METHOD PUBLIC ClearReference
VAR_INPUT
END_VAR
activeData REF= localData;
SetMemberReference();
END_METHOD

PROPERTY PUBLIC Size : UDINT
GET
Size := SIZEOF(activeData);
END_GET
END_PROPERTY

METHOD FB_init : BOOL
VAR_INPUT
	bInitRetains : BOOL; // if TRUE, the retain variables are initialized (warm start / cold start)
	bInCopyCode : BOOL;  // if TRUE, the instance afterwards gets moved into the copy code (online change)
END_VAR
SetMemberReference();
AddMember('bFilterByArea', _bFilterByArea);
AddMember('bFilterByCircularity', _bFilterByCircularity);
AddMember('bFilterByColor', _bFilterByColor);
AddMember('bFilterByConvexity', _bFilterByConvexity);
AddMember('bFilterByInertia', _bFilterByInertia);
AddMember('fMinArea', _fMinArea);
AddMember('fMaxArea', _fMaxArea);
AddMember('fMinCircularity', _fMinCircularity);
AddMember('fMaxCircularity', _fMaxCircularity);
AddMember('nBlobColor', _nBlobColor);
AddMember('fMinConvexity', _fMinConvexity);
AddMember('fMaxConvexity', _fMaxConvexity);
AddMember('fMinInertiaRatio', _fMinInertiaRatio);
AddMember('fMaxInertiaRatio', _fMaxInertiaRatio);
AddMember('fMinBlobDist', _fMinBlobDist);
AddMember('nMinRepeatability', _nMinRepeatability);
AddMember('fMinThreshold', _fMinThreshold);
AddMember('fMaxThreshold', _fMaxThreshold);
AddMember('fThresholdStep',  _fThresholdStep);
END_METHOD

METHOD PROTECTED SetMemberReference
VAR_INPUT
END_VAR
_bFilterByArea.MakeReferenceTo(activeData.bFilterByArea);
_bFilterByCircularity.MakeReferenceTo(activeData.bFilterByCircularity);
_bFilterByColor.MakeReferenceTo(activeData.bFilterByColor);
_bFilterByConvexity.MakeReferenceTo(activeData.bFilterByConvexity);
_bFilterByInertia.MakeReferenceTo(activeData.bFilterByInertia);
_fMinArea.MakeReferenceTo(activeData.fMinArea);
_fMaxArea.MakeReferenceTo(activeData.fMaxArea);
_fMinCircularity.MakeReferenceTo(activeData.fMinCircularity);
_fMaxCircularity.MakeReferenceTo(activeData.fMaxCircularity);
_nBlobColor.MakeReferenceTo(activeData.nBlobColor);
_fMinConvexity.MakeReferenceTo(activeData.fMinConvexity);
_fMaxConvexity.MakeReferenceTo(activeData.fMaxConvexity);
_fMinInertiaRatio.MakeReferenceTo(activeData.fMinInertiaRatio);
_fMaxInertiaRatio.MakeReferenceTo(activeData.fMaxInertiaRatio);
_fMinBlobDist.MakeReferenceTo(activeData.fMinBlobDist);
_nMinRepeatability.MakeReferenceTo(activeData.nMinRepeatability);
_fMinThreshold.MakeReferenceTo(activeData.fMinThreshold);
_fMaxThreshold.MakeReferenceTo(activeData.fMaxThreshold);
_fThresholdStep.MakeReferenceTo(activeData.fThresholdStep);
END_METHOD

METHOD PUBLIC Clone : I_Datatype
VAR
    pClone : POINTER TO _TcVnParamsSB;
END_VAR
pClone := __NEW(_TcVnParamsSB());
pClone^.Value := Value;
Clone := pClone^;
END_METHOD

PROPERTY PUBLIC Identifier : T_MAXSTRING
GET
Identifier := 'TcVnParamsSB';
END_GET
END_PROPERTY

METHOD PUBLIC MakeReferenceTo
VAR_INPUT
	ReferenceTarget : REFERENCE TO TcVnParamsSB;
END_VAR
activeData REF= ReferenceTarget;
SetMemberReference();
END_METHOD

METHOD TryMakeReferenceTo : BOOL
VAR_INPUT
	Target : I_Datatype;
END_VAR
VAR
	pTargetData : POINTER TO TcVnParamsSB;
END_VAR
IF NOT IsEquivalentTo(Target) THEN
	RETURN;
END_IF

pTargetData := Target.Address;
activeData REF= pTargetData^;
SetMemberReference();
TryMakeReferenceTo := TRUE;
END_METHOD

PROPERTY PUBLIC Value : REFERENCE TO TcVnParamsSB
GET
Value REF= activeData;
END_GET
END_PROPERTY

PROPERTY PUBLIC bFilterByArea : REFERENCE TO _BOOL
GET
bFilterByArea REF= _bFilterByArea;
END_GET
END_PROPERTY

PROPERTY PUBLIC bFilterByCircularity : REFERENCE TO _BOOL
GET
bFilterByCircularity REF= _bFilterByCircularity;
END_GET
END_PROPERTY

PROPERTY PUBLIC bFilterByColor : REFERENCE TO _BOOL
GET
bFilterByColor REF= _bFilterByColor;
END_GET
END_PROPERTY

PROPERTY PUBLIC bFilterByConvexity : REFERENCE TO _BOOL
GET
bFilterByConvexity REF= _bFilterByConvexity;
END_GET
END_PROPERTY

PROPERTY PUBLIC bFilterByInertia : REFERENCE TO _BOOL
GET
bFilterByInertia REF= _bFilterByInertia;
END_GET
END_PROPERTY

PROPERTY PUBLIC fMaxArea : REFERENCE TO _REAL
GET
fMaxArea REF= _fMaxArea;
END_GET
END_PROPERTY

PROPERTY PUBLIC fMaxCircularity : REFERENCE TO _REAL
GET
fMaxCircularity REF= _fMaxCircularity;
END_GET
END_PROPERTY

PROPERTY PUBLIC fMaxConvexity : REFERENCE TO _REAL
GET
fMaxConvexity REF= _fMaxConvexity;
END_GET
END_PROPERTY

PROPERTY PUBLIC fMaxInertiaRatio : REFERENCE TO _REAL
GET
fMaxInertiaRatio REF= _fMaxInertiaRatio;
END_GET
END_PROPERTY

PROPERTY PUBLIC fMaxThreshold : REFERENCE TO _REAL
GET
fMaxThreshold REF= _fMaxThreshold;
END_GET
END_PROPERTY

PROPERTY PUBLIC fMinArea : REFERENCE TO _REAL
GET
fMinArea REF= _fMinArea;
END_GET
END_PROPERTY

PROPERTY PUBLIC fMinBlobDist : REFERENCE TO _REAL
GET
fMinBlobDist REF= _fMinBlobDist;
END_GET
END_PROPERTY

PROPERTY PUBLIC fMinCircularity : REFERENCE TO _REAL
GET
fMinCircularity REF= _fMinCircularity;
END_GET
END_PROPERTY

PROPERTY PUBLIC fMinConvexity : REFERENCE TO _REAL
GET
fMinConvexity REF= _fMinConvexity;
END_GET
END_PROPERTY

PROPERTY PUBLIC fMinInertiaRatio : REFERENCE TO _REAL
GET
fMinInertiaRatio REF= _fMinInertiaRatio;
END_GET
END_PROPERTY

PROPERTY PUBLIC fMinThreshold : REFERENCE TO _REAL
GET
fMinThreshold REF= _fMinThreshold;
END_GET
END_PROPERTY

PROPERTY PUBLIC fThresholdStep : REFERENCE TO _REAL
GET
fThresholdStep REF= _fThresholdStep;
END_GET
END_PROPERTY

PROPERTY PUBLIC nBlobColor : REFERENCE TO _USINT
GET
nBlobColor REF= _nBlobColor;
END_GET
END_PROPERTY

PROPERTY PUBLIC nMinRepeatability : REFERENCE TO _UDINT
GET
nMinRepeatability REF= _nMinRepeatability;
END_GET
END_PROPERTY

END_FUNCTION_BLOCK

// Datatypes/Structs/_TcVnParamsWalshBarcodeDetection
{attribute 'linkalways'}
{attribute 'no_explicit_call' := 'This FB is a CLASS and must be accessed using methods or properties'}
{attribute 'enable_dynamic_creation'}
FUNCTION_BLOCK _TcVnParamsWalshBarcodeDetection EXTENDS StructuredDatatypeBase
VAR
    localData : TcVnParamsWalshBarcodeDetection := (nMaxBarDistance := 8, fMinAspectRatio := 1.0, fMaxAspectRatio := 5.0, nIntensityDifference := 100, nMinArea := -1, nChannelIndex := -1, nWalshFilterNum := 5, fOutlierReductionFactor := 1.0, fBarConnectionFactor := 1.0, fRegionFilterFactor := 1.0, fPostProcessingResizeFactor := 0.5, eInterpolationType := TCVN_IT_BILINEAR);
    activeData : REFERENCE TO TcVnParamsWalshBarcodeDetection REF= localData;
    _nMaxBarDistance : _UDINT(localData.nMaxBarDistance);
    _fMinAspectRatio : _REAL(localData.fMinAspectRatio);
    _fMaxAspectRatio : _REAL(localData.fMaxAspectRatio);
    _nIntensityDifference : _UDINT(localData.nIntensityDifference);
    _nMinArea : _DINT(localData.nMinArea);
    _nChannelIndex : _DINT(localData.nChannelIndex);
    _nWalshFilterNum : _UDINT(localData.nWalshFilterNum);
    _fOutlierReductionFactor : _REAL(localData.fOutlierReductionFactor);
    _fBarConnectionFactor : _REAL(localData.fBarConnectionFactor);
    _fRegionFilterFactor : _REAL(localData.fRegionFilterFactor);
    _fPostProcessingResizeFactor : _REAL(localData.fPostProcessingResizeFactor);
    _eInterpolationType : _ETcVnInterpolationType(localData.eInterpolationType);
END_VAR

PROPERTY PUBLIC Address : PVOID
GET
Address := ADR(activeData);
END_GET
END_PROPERTY

METHOD PUBLIC ClearReference
VAR_INPUT
END_VAR
activeData REF= localData;
SetMemberReference();
END_METHOD

PROPERTY PUBLIC Size : UDINT
GET
Size := SIZEOF(activeData);
END_GET
END_PROPERTY

METHOD FB_init : BOOL
VAR_INPUT
	bInitRetains : BOOL; // if TRUE, the retain variables are initialized (warm start / cold start)
	bInCopyCode : BOOL;  // if TRUE, the instance afterwards gets moved into the copy code (online change)
END_VAR
SetMemberReference();
AddMember('nMaxBarDistance', _nMaxBarDistance);
AddMember('fMinAspectRatio', _fMinAspectRatio);
AddMember('fMaxAspectRatio', _fMaxAspectRatio);
AddMember('nIntensityDifference', _nIntensityDifference);
AddMember('nMinArea', _nMinArea);
AddMember('nChannelIndex', _nChannelIndex);
AddMember('nWalshFilterNum', _nWalshFilterNum);
AddMember('fOutlierReductionFactor', _fOutlierReductionFactor);
AddMember('fBarConnectionFactor', _fBarConnectionFactor);
AddMember('fRegionFilterFactor', _fRegionFilterFactor);
AddMember('fPostProcessingResizeFactor', _fPostProcessingResizeFactor);
AddMember('eInterpolationType', _eInterpolationType);
END_METHOD

METHOD PROTECTED SetMemberReference
VAR_INPUT
END_VAR
_nMaxBarDistance.MakeReferenceTo(activeData.nMaxBarDistance);
_fMinAspectRatio.MakeReferenceTo(activeData.fMinAspectRatio);
_fMaxAspectRatio.MakeReferenceTo(activeData.fMaxAspectRatio);
_nIntensityDifference.MakeReferenceTo(activeData.nIntensityDifference);
_nMinArea.MakeReferenceTo(activeData.nMinArea);
_nChannelIndex.MakeReferenceTo(activeData.nChannelIndex);
_nWalshFilterNum.MakeReferenceTo(activeData.nWalshFilterNum);
_fOutlierReductionFactor.MakeReferenceTo(activeData.fOutlierReductionFactor);
_fBarConnectionFactor.MakeReferenceTo(activeData.fBarConnectionFactor);
_fRegionFilterFactor.MakeReferenceTo(activeData.fRegionFilterFactor);
_fPostProcessingResizeFactor.MakeReferenceTo(activeData.fPostProcessingResizeFactor);
_eInterpolationType.MakeReferenceTo(activeData.eInterpolationType);
END_METHOD

METHOD PUBLIC Clone : I_Datatype
VAR
    pClone : POINTER TO _TcVnParamsWalshBarcodeDetection;
END_VAR
pClone := __NEW(_TcVnParamsWalshBarcodeDetection);
IF pClone = 0 THEN
    RETURN;
END_IF
pClone^.TryCopyFrom(THIS^);
Clone := pClone^;
END_METHOD

PROPERTY PUBLIC Identifier : T_MAXSTRING
GET
Identifier := 'TcVnParamsWalshBarcodeDetection';
END_GET
END_PROPERTY

METHOD PUBLIC MakeReferenceTo
VAR_INPUT
	ReferenceTarget : REFERENCE TO TcVnParamsWalshBarcodeDetection;
END_VAR
activeData REF= ReferenceTarget;
SetMemberReference();
END_METHOD

METHOD TryMakeReferenceTo : BOOL
VAR_INPUT
	Target : I_Datatype;
END_VAR
VAR
	pTargetData : POINTER TO TcVnParamsWalshBarcodeDetection;
END_VAR
IF NOT IsEquivalentTo(Target) THEN
	RETURN;
END_IF

pTargetData := Target.Address;
activeData REF= pTargetData^;
SetMemberReference();
TryMakeReferenceTo := TRUE;
END_METHOD

PROPERTY PUBLIC Value : REFERENCE TO TcVnParamsWalshBarcodeDetection
GET
Value REF= activeData;
END_GET
END_PROPERTY

PROPERTY PUBLIC eInterpolationType : REFERENCE TO _ETcVnInterpolationType
GET
eInterpolationType REF= _eInterpolationType;
END_GET
END_PROPERTY

PROPERTY PUBLIC fBarConnectionFactor : REFERENCE TO _REAL
GET
fBarConnectionFactor REF= _fBarConnectionFactor;
END_GET
END_PROPERTY

PROPERTY PUBLIC fMaxAspectRatio : REFERENCE TO _REAL
GET
fMaxAspectRatio REF= _fMaxAspectRatio;
END_GET
END_PROPERTY

PROPERTY PUBLIC fMinAspectRatio : REFERENCE TO _REAL
GET
fMinAspectRatio REF= _fMinAspectRatio;
END_GET
END_PROPERTY

PROPERTY PUBLIC fOutlierReductionFactor : REFERENCE TO _REAL
GET
fOutlierReductionFactor REF= _fOutlierReductionFactor;
END_GET
END_PROPERTY

PROPERTY PUBLIC fPostProcessingResizeFactor : REFERENCE TO _REAL
GET
fPostProcessingResizeFactor REF= _fPostProcessingResizeFactor;
END_GET
END_PROPERTY

PROPERTY PUBLIC fRegionFilterFactor : REFERENCE TO _REAL
GET
fRegionFilterFactor REF= _fRegionFilterFactor;
END_GET
END_PROPERTY

PROPERTY PUBLIC nChannelIndex : REFERENCE TO _DINT
GET
nChannelIndex REF= _nChannelIndex;
END_GET
END_PROPERTY

PROPERTY PUBLIC nIntensityDifference : REFERENCE TO _UDINT
GET
nIntensityDifference REF= _nIntensityDifference;
END_GET
END_PROPERTY

PROPERTY PUBLIC nMaxBarDistance : REFERENCE TO _UDINT
GET
nMaxBarDistance REF= _nMaxBarDistance;
END_GET
END_PROPERTY

PROPERTY PUBLIC nMinArea : REFERENCE TO _DINT
GET
nMinArea REF= _nMinArea;
END_GET
END_PROPERTY

PROPERTY PUBLIC nWalshFilterNum : REFERENCE TO _UDINT
GET
nWalshFilterNum REF= _nWalshFilterNum;
END_GET
END_PROPERTY

END_FUNCTION_BLOCK

// Datatypes/Structs/_TcVnRectangle_UDINT
{attribute 'linkalways'} 
{attribute 'no_explicit_call' := 'This FB is a CLASS and must be accessed using methods or properties'}
{attribute 'enable_dynamic_creation'}
FUNCTION_BLOCK _TcVnRectangle_UDINT EXTENDS StructuredDatatypeBase
VAR
	localData : TcVnRectangle_UDINT;
	activeData : REFERENCE TO TcVnRectangle_UDINT REF= localData;
	_nX : _UDINT(localData.nX);
	_nY : _UDINT(localData.nY);
    _nWidth : _UDINT(localData.nWidth);
	_nHeight : _UDINT(localData.nHeight);
END_VAR

PROPERTY PUBLIC Address : PVOID
GET
Address := ADR(activeData);
END_GET
END_PROPERTY

METHOD PUBLIC ClearReference
VAR_INPUT
END_VAR
activeData REF= localData;
SetMemberReference();
END_METHOD

PROPERTY PUBLIC Size : UDINT
GET
Size := SIZEOF(activeData);
END_GET
END_PROPERTY

METHOD FB_init : BOOL
VAR_INPUT
	bInitRetains : BOOL; // if TRUE, the retain variables are initialized (warm start / cold start)
	bInCopyCode : BOOL;  // if TRUE, the instance afterwards gets moved into the copy code (online change)
END_VAR
SetMemberReference();
AddMember('nX',_nX);
AddMember('nY',_nY);
AddMember('nWidth',_nWidth);
AddMember('nHeight',_nHeight);
END_METHOD

METHOD PROTECTED SetMemberReference
VAR_INPUT
END_VAR
_nX.MakeReferenceTo(activeData.nX);
_nY.MakeReferenceTo(activeData.nY);
_nWidth.MakeReferenceTo(activeData.nWidth);
_nHeight.MakeReferenceTo(activeData.nHeight);
END_METHOD

METHOD PUBLIC Clone : I_Datatype
VAR
    pClone : POINTER TO _TcVnRectangle_UDINT;
END_VAR
pClone := __NEW(_TcVnRectangle_UDINT());
pClone^.Value := Value;
Clone := pClone^;
END_METHOD

PROPERTY PUBLIC Identifier : T_MAXSTRING
GET
Identifier := 'TcVnRectangle_UDINT';
END_GET
END_PROPERTY

METHOD PUBLIC MakeReferenceTo
VAR_INPUT
	ReferenceTarget : REFERENCE TO TcVnRectangle_UDINT;
END_VAR
activeData REF= ReferenceTarget;
SetMemberReference();
END_METHOD

METHOD TryMakeReferenceTo : BOOL
VAR_INPUT
	Target : I_Datatype;
END_VAR
VAR
	pTargetData : POINTER TO TcVnRectangle_UDINT;
END_VAR
IF NOT IsEquivalentTo(Target) THEN
	RETURN;
END_IF

pTargetData := Target.Address;
activeData REF= pTargetData^;
SetMemberReference();
TryMakeReferenceTo := TRUE;
END_METHOD

PROPERTY PUBLIC Value : REFERENCE TO TcVnRectangle_UDINT
GET
Value REF= activeData;
END_GET
END_PROPERTY

PROPERTY PUBLIC nHeight : REFERENCE TO _UDINT
GET
nHeight REF= _nHeight;
END_GET
END_PROPERTY

PROPERTY PUBLIC nWidth : REFERENCE TO _UDINT
GET
nWidth REF= _nWidth;
END_GET
END_PROPERTY

PROPERTY PUBLIC nX : REFERENCE TO _UDINT
GET
nX REF= _nX;
END_GET
END_PROPERTY

PROPERTY PUBLIC nY : REFERENCE TO _UDINT
GET
nY REF= _nY;
END_GET
END_PROPERTY

END_FUNCTION_BLOCK

// Datatypes/VisionDatatypePack
{attribute 'linkalways'} 
{attribute 'no_explicit_call' := 'This FB is a CLASS and must be accessed using methods or properties'}
{attribute 'enable_dynamic_creation'}
FUNCTION_BLOCK VisionDatatypePack
VAR
    // aliases
    _gVCP_REGISTER_ADDRESS : _GVCP_REGISTER_ADDRESS(0);
    _gVCP_REGISTER_VALUE : _GVCP_REGISTER_VALUE(0);
    _tcVnPoint : _TcVnPoint;
    _tcVnPoint2_DINT : _TcVnPoint2_DINT;
    _tcVnPoint2_LREAL : _TcVnPoint2_LREAL;
    _tcVnPoint2_REAL : _TcVnPoint2_REAL;
    _tcVnPoint3_LREAL : _TcVnPoint3_LREAL;
    _tcVnPoint3_REAL : _TcVnPoint3_REAL;
    _tcVnRectangle : _TcVnRectangle;
  
    _tcVnArray10_ITcVnImage : _TcVnArray10_ITcVnImage;
    _tcVnArray3_Point2_REAL : _TcVnArray3_Point2_REAL;
    _tcVnArray33_UDINT : _TcVnArray33_UDINT;
    _tcVnArray4_LREAL : _TcVnArray4_LREAL;
    _tcVnArray4_Point2_REAL : _TcVnArray4_Point2_REAL;
    _tcVnArray7_LREAL : _TcVnArray7_LREAL;
    _tcVnArray8_LREAL : _TcVnArray8_LREAL;
    _tcVnMatrix2x3_LREAL : _TcVnMatrix2x3_LREAL;
    _tcVnMatrix3x3_LREAL : _TcVnMatrix3x3_LREAL;
    _tcVnVector2_DINT : _TcVnVector2_DINT;
    _tcVnVector2_INT : _TcVnVector2_INT;
    _tcVnVector2_LREAL : _TcVnVector2_LREAL;
    _tcVnVector2_REAL : _TcVnVector2_REAL;
    _tcVnVector2_SINT : _TcVnVector2_SINT;
    _tcVnVector2_UINT : _TcVnVector2_UINT;
    _tcVnVector2_USINT : _TcVnVector2_USINT;
    _tcVnVector3_INT : _TcVnVector3_INT;
    _tcVnVector3_LREAL : _TcVnVector3_LREAL;
    _tcVnVector3_REAL : _TcVnVector3_REAL;
    _tcVnVector3_SINT : _TcVnVector3_SINT;
    _tcVnVector3_UINT : _TcVnVector3_UINT;
    _tcVnVector3_USINT : _TcVnVector3_USINT;
    _tcVnVector4_DINT : _TcVnVector4_DINT;
    _tcVnVector4_INT : _TcVnVector4_INT;
    _tcVnVector4_LREAL : _TcVnVector4_LREAL;
    _tcVnVector4_REAL : _TcVnVector4_REAL;
    _tcVnVector4_SINT : _TcVnVector4_SINT;
    _tcVnVector4_UINT : _TcVnVector4_UINT;
    _tcVnVector4_USINT : _TcVnVector4_USINT;
 
    // constants
    
    // arrays
    _array0to1OfDINT : _Array0to1OfDINT;
    _array0to1OfINT : _Array0to1OfINT;
    _array0to1OfLREAL : _Array0to1OfLREAL;
    _array0to1OfREAL : _Array0to1OfREAL;
    _array0to1OfSINT : _Array0to1OfSINT;
    _array0to1OfUINT : _Array0to1OfUINT;
    _array0to1OfUSINT : _Array0to1OfUSINT;
    _array0to2OfINT : _Array0to2OfINT;
    _array0to2OfLREAL : _Array0to2OfLREAL;
    _array0to2OfREAL : _Array0to2OfREAL;
    _array0to2OfSINT : _Array0to2OfSINT;
    _array0to2OfUINT : _Array0to2OfUINT;
    _array0to2OfUSINT : _Array0to2OfUSINT;
    _array0to3OfDINT : _Array0to3OfDINT;
    _array0to3OfINT : _Array0to3OfINT;
	_array0to3OfLREAL : _Array0to3OfLREAL;
    _array0to3OfREAL : _Array0to3OfREAL;
    _array0to6OfLREAL : _Array0to6OfLREAL;
    _array0to7OfLREAL : _Array0to7OfLREAL;
	_array0to1_0to2OfLREAL : _Array0to1_0to2OfLREAL;
	_array0to2_0to2OfLREAL : _Array0to2_0to2OfLREAL;
    
    // enums
	_eTcVn2dCodeSearchStrategy : _ETcVn2dCodeSearchStrategy(ETcVn2dCodeSearchStrategy.TCVN_CSS_DEFAULT);
    _eTcVnAdaptiveThresholdMethod : _ETcVnAdaptiveThresholdMethod(ETcVnAdaptiveThresholdMethod.TCVN_ATM_MEAN);
    _eTcVnBarcodeSearchDirection : _ETcVnBarcodeSearchDirection(ETcVnBarcodeSearchDirection.TCVN_BSD_ANY);
    _eTcVnBarcodeType : _ETcVnBarcodeType(ETcVnBarcodeType.TCVN_BT_CODABAR);
    _eTcVnBlobCombination : _ETcVnBlobCombination(ETcVnBlobCombination.TCVN_BC_SMALLEST);
    _eTcVnBoostClassifierType : _ETcVnBoostClassifierType(ETcVnBoostClassifierType.TCVN_BCT_DISCRETE);
    _eTcVnBorderInterpolationMethod : _ETcVnBorderInterpolationMethod(ETcVnBorderInterpolationMethod.TCVN_BIM_DEFAULT);
    _eTcVnCalibrationPattern : _ETcVnCalibrationPattern(ETcVnCalibrationPattern.TCVN_CP_CIRCLES_SYM);
    _eTcVnCalibrationPatternOrigin : _ETcVnCalibrationPatternOrigin(ETcVnCalibrationPatternOrigin.TCVN_CPO_TOPCENTER);
    _eTcVnCameraState : _ETcVnCameraState(ETcVnCameraState.TCVN_CS_INITIAL);
    _eTcVnClusteringAlgorithm : _ETcVnClusteringAlgorithm(ETcVnClusteringAlgorithm.TCVN_CA_KMEANSPP);
	_eTcVnCodeDetectionModel : _ETcVnCodeDetectionModel(ETcVnCodeDetectionModel.TCVN_CDM_DETECT_1_1);
	_eTcVnCodeType : _ETcVnCodeType(ETcVnCodeType.TCVN_CT_ANY);
    _eTcVnColorMap : _ETcVnColorMap(ETcVnColorMap.TCVN_CM_AUTUMN);
    _eTcVnColorMapSize : _ETcVnColorMapSize(ETcVnColorMapSize.TCVN_CMS_256);
    _eTcVnColorSpaceTransform : _ETcVnColorSpaceTransform(ETcVnColorSpaceTransform.TCVN_CST_RGBA_TO_RGB);
    _eTcVnColorTrainingMethod : _ETcVnColorTrainingMethod(ETcVnColorTrainingMethod.TCVN_CTM_LAB);
    _eTcVnConnectedComponentsAlgorithm : _ETcVnConnectedComponentsAlgorithm(ETcVnConnectedComponentsAlgorithm.TCVN_CCA_WU);
    _eTcVnContainerExportFormat : _ETcVnContainerExportFormat(ETcVnContainerExportFormat.TCVN_CEF_XML);
    _eTcVnContourApproximationMethod : _ETcVnContourApproximationMethod(ETcVnContourApproximationMethod.TCVN_CAM_NONE);
    _eTcVnContourRetrievalMode : _ETcVnContourRetrievalMode(ETcVnContourRetrievalMode.TCVN_CRM_EXTERNAL);
    _eTcVnContoursMatchComparisonMethod : _ETcVnContoursMatchComparisonMethod(ETcVnContoursMatchComparisonMethod.TCVN_CMCM_CONTOURS_MATCH_I1);
    _eTcVnDiffusivityTypeKAZE : _ETcVnDiffusivityTypeKAZE(ETcVnDiffusivityTypeKAZE.TCVN_DT1_KAZE_PM_G1);
    _eTcVnDistanceTransformationLabel : _ETcVnDistanceTransformationLabel(ETcVnDistanceTransformationLabel.TCVN_DTL_CCOMP);
    _eTcVnDistanceTransformationMask : _ETcVnDistanceTransformationMask(ETcVnDistanceTransformationMask.TCVN_DTM_PRECISE);
    _eTcVnDistanceType : _ETcVnDistanceType(ETcVnDistanceType.TCVN_DT_USER);
    _eTcVnDrawMatchesFlags : _ETcVnDrawMatchesFlags(ETcVnDrawMatchesFlags.TCVN_DMF_DEFAULT);
    _eTcVnDrawShape : _ETcVnDrawShape(ETcVnDrawShape.TCVN_DS_CIRCLE);
    _eTcVnEdgeDetectionAlgorithm : _ETcVnEdgeDetectionAlgorithm(ETcVnEdgeDetectionAlgorithm.TCVN_EDA_INTERPOLATION);
    _eTcVnEdgeDirection : _ETcVnEdgeDirection(ETcVnEdgeDirection.TCVN_ED_DARK_TO_LIGHT);
    _eTcVnElementType : _ETcVnElementType(ETcVnElementType.TCVN_ET_SAME_AS_SOURCE);
    _eTcVnEstimationAlgorithm : _ETcVnEstimationAlgorithm(ETcVnEstimationAlgorithm.TCVN_EA_DEFAULT);
    _eTcVnExtremePointDirection : _ETcVnExtremePointDirection(ETcVnExtremePointDirection.TCVN_EPD_TOP_LEFT);
    _eTcVnFeatureDescriptorTypeAKAZE : _ETcVnFeatureDescriptorTypeAKAZE(ETcVnFeatureDescriptorTypeAKAZE.TCVN_FDT_AKAZE_KAZE_UPRIGHT);
    _eTcVnFeatureScalingType : _ETcVnFeatureScalingType(ETcVnFeatureScalingType.TCVN_FST1_MAXABS);
    _eTcVnFeatureScoreTypeORB : _ETcVnFeatureScoreTypeORB(ETcVnFeatureScoreTypeORB.TCVN_FST_ORB_HARRIS);
    _eTcVnFilterDirection : _ETcVnFilterDirection(ETcVnFilterDirection.TCVN_FD_X);
	_eTcVnFindTemplateWalshOptions : _ETcVnFindTemplateWalshOptions(ETcVnFindTemplateWalshOptions.TCVN_FTWO_NONE);
    _eTcVnFlipAxis : _ETcVnFlipAxis(ETcVnFlipAxis.TCVN_FA_X);
    _eTcVnFontType : _ETcVnFontType(ETcVnFontType.TCVN_FT_HERSHEY_SIMPLEX);
    _eTcVnHoughMethod : _ETcVnHoughMethod(ETcVnHoughMethod.TCVN_HM_STANDARD);
    _eTcVnInitializableFunction : _ETcVnInitializableFunction(ETcVnInitializableFunction.TCVN_IF_OCR);
    _eTcVnInterpolationType : _ETcVnInterpolationType(ETcVnInterpolationType.TCVN_IT_NEAREST_NEIGHBOR);
    _eTcVnKeypointDetectionTypeAGAST : _ETcVnKeypointDetectionTypeAGAST(ETcVnKeypointDetectionTypeAGAST.TCVN_KDT_AGAST_5_8);
    _eTcVnKeypointDetectionTypeFAST : _ETcVnKeypointDetectionTypeFAST(ETcVnKeypointDetectionTypeFAST.TCVN_KDT_FAST_5_8);
    _eTcVnKnn : _ETcVnKnn(ETcVnKnn.TCVN_KNN_CLASSIFIER);
    _eTcVnLineType : _ETcVnLineType(ETcVnLineType.TCVN_LT_4_CONNECTED);
	_eTcVnMatchTemplateWalshOptions : _ETcVnMatchTemplateWalshOptions(ETcVnMatchTemplateWalshOptions.TCVN_MTWO_NONE);
    _eTcVnMorphologicalOperator : _ETcVnMorphologicalOperator(ETcVnMorphologicalOperator.TCVN_MO_EROSION);
    _eTcVnNbc : _ETcVnNbc(ETcVnNbc.TCVN_NBC_CLASSIFIER);
    _eTcVnNormalizationType : _ETcVnNormalizationType(ETcVnNormalizationType.TCVN_NT_INF);
    _eTcVnOcrModelType : _ETcVnOcrModelType(ETcVnOcrModelType.TCVN_OMT_NUMBERS);
    _eTcVnOcrOptions : _ETcVnOcrOptions(ETcVnOcrOptions.TCVN_OO_NONE);
    _eTcVnOrientationMethod : _ETcVnOrientationMethod(ETcVnOrientationMethod.TCVN_OM_PCA);
    _eTcVnPaddingMode : _ETcVnPaddingMode(ETcVnPaddingMode.TCVN_PM_NONE);
    _eTcVnPixelConnectivity : _ETcVnPixelConnectivity(ETcVnPixelConnectivity.TCVN_PC_4);
    _eTcVnPixelEncoding : _ETcVnPixelEncoding(ETcVnPixelEncoding.TCVN_PE_NONE);
    _eTcVnPixelPackMode : _ETcVnPixelPackMode(ETcVnPixelPackMode.TCVN_PPM_NONE);
    _eTcVnPrototypeClusterer : _ETcVnPrototypeClusterer(ETcVnPrototypeClusterer.TCVN_PC_NOVELTY_DETECTOR);
    _eTcVnRectangleIntersection : _ETcVnRectangleIntersection(ETcVnRectangleIntersection.TCVN_RI_NONE);
    _eTcVnRotationAngle : _ETcVnRotationAngle(ETcVnRotationAngle.TCVN_RA_90_DEG);
    _eTcVnRTrees : _ETcVnRTrees(ETcVnRTrees.TCVN_RT_CLASSIFIER);
    _eTcVnSignedNormalization : _ETcVnSignedNormalization(ETcVnSignedNormalization.TCVN_SN_FIX_ZERO);
    _eTcVnSolvePnPMethod : _ETcVnSolvePnPMethod(ETcVnSolvePnPMethod.TCVN_SPM_ITERATIVE);
    _eTcVnSta : _ETcVnSta(ETcVnSta.TCVN_STA_CLASSIFIER);
    _eTcVnStructuringElementShape : _ETcVnStructuringElementShape(ETcVnStructuringElementShape.TCVN_SES_RECTANGLE);
    _eTcVnSvm : _ETcVnSvm(ETcVnSvm.TCVN_SVM_C_CLASSIFIER);
    _eTcVnSvmKernelType : _ETcVnSvmKernelType(ETcVnSvmKernelType.TCVN_SKT_LINEAR);
    _eTcVnSvmSgdClassifierMarginType : _ETcVnSvmSgdClassifierMarginType(ETcVnSvmSgdClassifierMarginType.TCVN_SSCMT_SOFT_MARGIN);
    _eTcVnSvmSgdClassifierType : _ETcVnSvmSgdClassifierType(ETcVnSvmSgdClassifierType.TCVN_SSCT_SGD);
    _eTcVnTemplateMatchMethod : _ETcVnTemplateMatchMethod(ETcVnTemplateMatchMethod.TCVN_TMM_SQDIFF);
    _eTcVnThresholdType : _ETcVnThresholdType(ETcVnThresholdType.TCVN_TT_BINARY);
    _eTcVnTimestamp : _ETcVnTimestamp(ETcVnTimestamp.TCVN_TS_IMAGE_COMPLETED);
    _eTcVnVectorCompareMethod : _ETcVnVectorCompareMethod(ETcVnVectorCompareMethod.TCVN_VCM_EUCLIDEAN);
    _eTcVnWorldCoordinateSystem : _ETcVnWorldCoordinateSystem(ETcVnWorldCoordinateSystem.TCVN_WCS_X_RIGHT_Y_DOWN);
    _eTcWatchdogAccumulationType : _ETcWatchdogAccumulationType(ETcWatchdogAccumulationType.WD_ACC_TYPE_MEAN);
    _gEV_CAMERA_STATE : _GEV_CAMERA_STATE(GEV_CAMERA_STATE.GEV_CAMERA_IDLE);
    _eTcVnDataLayout : _ETcVnDataLayout(ETcVnDataLayout.TCVN_DL_DEFAULT);
    _eTcVnReduceType : _ETcVnReduceType(ETcVnReduceType.TCVN_RT_REDUCE_SUM);
    _eTcVnCircularityCalculationMethod : _ETcVnCircularityCalculationMethod(ETcVnCircularityCalculationMethod.TCVN_CCM_DEFAULT);
    _eTcVnDataMatrixOptions : _ETcVnDataMatrixOptions(ETcVnDataMatrixOptions.TCVN_DMO_DEFAULT);
    _eTcVnLayerNameType : _ETcVnLayerNameType(ETcVnLayerNameType.TCVN_LNT_ALL);
	
    _eTcVnComparisonOperator : _ETcVnComparisonOperator(ETcVnComparisonOperator.TCVN_CO_LESS);
    _eTcVnDetectBarcodesWalshOptions : _ETcVnDetectBarcodesWalshOptions(ETcVnDetectBarcodesWalshOptions.TCVN_DBWO_HORIZONTAL);
    _eTcVnDetectPatternPointsOptions : _ETcVnDetectPatternPointsOptions(ETcVnDetectPatternPointsOptions.TCVN_DPPO_SYMMETRIC);
    _eTcVnDotCodeOptions : _ETcVnDotCodeOptions(ETcVnDotCodeOptions.TCVN_DCO_DEFAULT);
    _eTcVnEdgeSelection : _ETcVnEdgeSelection(ETcVnEdgeSelection.TCVN_ES_RISING);
    _eTcVnFindRoisMethod : _ETcVnFindRoisMethod(ETcVnFindRoisMethod.TCVN_FRM_GRID);
    _eTcVnJpegSampling : _ETcVnJpegSampling(ETcVnJpegSampling.TCVN_JS_444);
    _eTcVnMergeRegionsOptions : _ETcVnMergeRegionsOptions(ETcVnMergeRegionsOptions.TCVN_MRO_UPRIGHT_BOUNDING_RECT);
    _eTcVnPolarizedImageInterpolation : _ETcVnPolarizedImageInterpolation(ETcVnPolarizedImageInterpolation.TCVN_PII_NONE);
    _eTcVnSalientFeaturesMethod : _ETcVnSalientFeaturesMethod(ETcVnSalientFeaturesMethod.TCVN_SFM_WALSH_CODE);
    // structs
    _gVSP_IMAGE_INFO : _GVSP_IMAGE_INFO;
    _gVSP_LEADER_PAYLOAD_IMAGE : _GVSP_LEADER_PAYLOAD_IMAGE;
    _gVSP_PIXEL_FORMAT : _GVSP_PIXEL_FORMAT;
    _tcVnCameraCalibrationOptions : _TcVnCameraCalibrationOptions;
    _tcVnCircularArc : _TcVnCircularArc;
    _tcVnCodeGrades1D : _TcVnCodeGrades1D;
    _tcVnCodeGradesDM : _TcVnCodeGradesDM;
    _tcVnCodeGradesQR : _TcVnCodeGradesQR;
    _tcVnDMatch : _TcVnDMatch;
	_tcVnImageInfo : _TcVnImageInfo;
    _tcVnKeyPoint : _TcVnKeyPoint;
//  _tcVnMatrix : _TcVnMatrix;
    _tcVnMoments : _TcVnMoments;
    _tcVnParamsAGAST : _TcVnParamsAGAST;
    _tcVnParamsAKAZE : _TcVnParamsAKAZE;
    _tcVnParamsBlobDetection : _TcVnParamsBlobDetection;
    _tcVnParamsBRISK : _TcVnParamsBRISK;
    _tcVnParamsFAST : _TcVnParamsFAST;
    _tcVnParamsGFTT : _TcVnParamsGFTT;
    _tcVnParamsKAZE : _TcVnParamsKAZE;
    _tcVnParamsMSER : _TcVnParamsMSER;
    _tcVnParamsORB : _TcVnParamsORB;
    _tcVnParamsSB : _TcVnParamsSB;
    _tcVnPixelFormat : _TcVnPixelFormat;
	_tcVnRectangle_DINT : _TcVnRectangle_DINT;
    _tcVnRectangle_UDINT : _TcVnRectangle_UDINT;
    _tcVnRotatedRectangle : _TcVnRotatedRectangle;
    _tcVnSize2_REAL : _TcVnSize2_REAL;
	
    _gVCP_ADDRESS_VALUE_PAIR : _GVCP_ADDRESS_VALUE_PAIR;
    _tcVnSize2_DINT : _TcVnSize2_DINT;
    _tcVnParamsFindRois : _TcVnParamsFindRois;
    _tcVnParamsWalshBarcodeDetection : _TcVnParamsWalshBarcodeDetection;
	// interfaces
	_iTcVnImage : _ITcVnImage;
	_iTcVnContainer : _ITcVnContainer;
	_iTcVnDisplayableImage : _ITcVnDisplayableImage;
	
END_VAR

METHOD RegisterWithDatatypes
VAR_INPUT
	Datatypes : I_Datatypes;
END_VAR
// aliases
Datatypes.RegisterDatatype(_GVCP_REGISTER_ADDRESS);
Datatypes.RegisterDatatype(_gVCP_REGISTER_VALUE);
Datatypes.RegisterDatatype(_tcVnPoint);
Datatypes.RegisterDatatype(_tcVnPoint2_DINT);
Datatypes.RegisterDatatype(_tcVnPoint2_LREAL);
Datatypes.RegisterDatatype(_tcVnPoint2_REAL);
Datatypes.RegisterDatatype(_tcVnPoint3_LREAL);
Datatypes.RegisterDatatype(_tcVnPoint3_REAL);
Datatypes.RegisterDatatype(_tcVnRectangle);

Datatypes.RegisterDatatype(_tcVnArray10_ITcVnImage);
Datatypes.RegisterDatatype(_tcVnArray3_Point2_REAL);
Datatypes.RegisterDatatype(_tcVnArray33_UDINT);
Datatypes.RegisterDatatype(_tcVnArray4_LREAL);
Datatypes.RegisterDatatype(_tcVnArray4_Point2_REAL);
Datatypes.RegisterDatatype(_tcVnArray7_LREAL);
Datatypes.RegisterDatatype(_tcVnArray8_LREAL);
Datatypes.RegisterDatatype(_tcVnMatrix2x3_LREAL);
Datatypes.RegisterDatatype(_tcVnMatrix3x3_LREAL);
Datatypes.RegisterDatatype(_tcVnVector2_DINT);
Datatypes.RegisterDatatype(_tcVnVector2_INT);
Datatypes.RegisterDatatype(_tcVnVector2_LREAL);
Datatypes.RegisterDatatype(_tcVnVector2_REAL);
Datatypes.RegisterDatatype(_tcVnVector2_SINT);
Datatypes.RegisterDatatype(_tcVnVector2_UINT);
Datatypes.RegisterDatatype(_tcVnVector2_USINT);
Datatypes.RegisterDatatype(_tcVnVector3_INT);
Datatypes.RegisterDatatype(_tcVnVector3_LREAL);
Datatypes.RegisterDatatype(_tcVnVector3_REAL);
Datatypes.RegisterDatatype(_tcVnVector3_SINT);
Datatypes.RegisterDatatype(_tcVnVector3_UINT);
Datatypes.RegisterDatatype(_tcVnVector3_USINT);
Datatypes.RegisterDatatype(_tcVnVector4_DINT);
Datatypes.RegisterDatatype(_tcVnVector4_INT);
Datatypes.RegisterDatatype(_tcVnVector4_LREAL);
Datatypes.RegisterDatatype(_tcVnVector4_REAL);
Datatypes.RegisterDatatype(_tcVnVector4_SINT);
Datatypes.RegisterDatatype(_tcVnVector4_UINT);
Datatypes.RegisterDatatype(_tcVnVector4_USINT);

// constants

// arrays
Datatypes.RegisterDatatype(_array0to1OfDINT);
Datatypes.RegisterDatatype(_array0to1OfINT);
Datatypes.RegisterDatatype(_array0to1OfLREAL);
Datatypes.RegisterDatatype(_array0to1OfREAL);
Datatypes.RegisterDatatype(_array0to1OfSINT);
Datatypes.RegisterDatatype(_array0to1OfUINT);
Datatypes.RegisterDatatype(_array0to1OfUSINT);
Datatypes.RegisterDatatype(_array0to2OfINT);
Datatypes.RegisterDatatype(_array0to2OfLREAL);
Datatypes.RegisterDatatype(_array0to2OfREAL);
Datatypes.RegisterDatatype(_array0to2OfSINT);
Datatypes.RegisterDatatype(_array0to2OfUINT);
Datatypes.RegisterDatatype(_array0to2OfUSINT);
Datatypes.RegisterDatatype(_array0to3OfDINT);
Datatypes.RegisterDatatype(_array0to3OfINT);
Datatypes.RegisterDatatype(_array0to3OfLREAL);
Datatypes.RegisterDatatype(_array0to3OfREAL);
Datatypes.RegisterDatatype(_array0to6OfLREAL);
Datatypes.RegisterDatatype(_array0to7OfLREAL);
Datatypes.RegisterDatatype(_array0to1_0to2OfLREAL);
Datatypes.RegisterDatatype(_array0to2_0to2OfLREAL);

// enums
Datatypes.RegisterDatatype(_eTcVn2dCodeSearchStrategy);
Datatypes.RegisterDatatype(_eTcVnAdaptiveThresholdMethod);
Datatypes.RegisterDatatype(_eTcVnBarcodeSearchDirection);
Datatypes.RegisterDatatype(_eTcVnBarcodeType);
Datatypes.RegisterDatatype(_eTcVnBlobCombination);
Datatypes.RegisterDatatype(_eTcVnBoostClassifierType);
Datatypes.RegisterDatatype(_eTcVnBorderInterpolationMethod);
Datatypes.RegisterDatatype(_eTcVnCalibrationPattern);
Datatypes.RegisterDatatype(_eTcVnCalibrationPatternOrigin);
Datatypes.RegisterDatatype(_eTcVnCameraState);
Datatypes.RegisterDatatype(_eTcVnClusteringAlgorithm);
Datatypes.RegisterDatatype(_eTcVnCodeDetectionModel);
Datatypes.RegisterDatatype(_eTcVnCodeType);
Datatypes.RegisterDatatype(_eTcVnColorMap);
Datatypes.RegisterDatatype(_eTcVnColorMapSize);
Datatypes.RegisterDatatype(_eTcVnColorSpaceTransform);
Datatypes.RegisterDatatype(_eTcVnColorTrainingMethod);
Datatypes.RegisterDatatype(_eTcVnConnectedComponentsAlgorithm);
Datatypes.RegisterDatatype(_eTcVnContainerExportFormat);
Datatypes.RegisterDatatype(_eTcVnContourApproximationMethod);
Datatypes.RegisterDatatype(_eTcVnContourRetrievalMode);
Datatypes.RegisterDatatype(_eTcVnContoursMatchComparisonMethod);
Datatypes.RegisterDatatype(_eTcVnDiffusivityTypeKAZE);
Datatypes.RegisterDatatype(_eTcVnDistanceTransformationLabel);
Datatypes.RegisterDatatype(_eTcVnDistanceTransformationMask);
Datatypes.RegisterDatatype(_eTcVnDistanceType);
Datatypes.RegisterDatatype(_eTcVnDrawMatchesFlags);
Datatypes.RegisterDatatype(_eTcVnDrawShape);
Datatypes.RegisterDatatype(_eTcVnEdgeDetectionAlgorithm);
Datatypes.RegisterDatatype(_eTcVnEdgeDirection);
Datatypes.RegisterDatatype(_eTcVnElementType);
Datatypes.RegisterDatatype(_eTcVnEstimationAlgorithm);
Datatypes.RegisterDatatype(_eTcVnExtremePointDirection);
Datatypes.RegisterDatatype(_eTcVnFeatureDescriptorTypeAKAZE);
Datatypes.RegisterDatatype(_eTcVnFeatureScalingType);
Datatypes.RegisterDatatype(_eTcVnFeatureScoreTypeORB);
Datatypes.RegisterDatatype(_eTcVnFilterDirection);
Datatypes.RegisterDatatype(_eTcVnFindTemplateWalshOptions);
Datatypes.RegisterDatatype(_eTcVnFlipAxis);
Datatypes.RegisterDatatype(_eTcVnFontType);
Datatypes.RegisterDatatype(_eTcVnHoughMethod);
Datatypes.RegisterDatatype(_eTcVnInitializableFunction);
Datatypes.RegisterDatatype(_eTcVnInterpolationType);
Datatypes.RegisterDatatype(_eTcVnKeypointDetectionTypeAGAST);
Datatypes.RegisterDatatype(_eTcVnKeypointDetectionTypeFAST);
Datatypes.RegisterDatatype(_eTcVnKnn);
Datatypes.RegisterDatatype(_eTcVnLineType);
Datatypes.RegisterDatatype(_eTcVnMatchTemplateWalshOptions);
Datatypes.RegisterDatatype(_eTcVnMorphologicalOperator);
Datatypes.RegisterDatatype(_eTcVnNbc);
Datatypes.RegisterDatatype(_eTcVnNormalizationType);
Datatypes.RegisterDatatype(_eTcVnOcrModelType);
Datatypes.RegisterDatatype(_eTcVnOcrOptions);
Datatypes.RegisterDatatype(_eTcVnOrientationMethod);
Datatypes.RegisterDatatype(_eTcVnPaddingMode);
Datatypes.RegisterDatatype(_eTcVnPixelConnectivity);
Datatypes.RegisterDatatype(_eTcVnPixelEncoding);
Datatypes.RegisterDatatype(_eTcVnPixelPackMode);
Datatypes.RegisterDatatype(_eTcVnPrototypeClusterer);
Datatypes.RegisterDatatype(_eTcVnRectangleIntersection);
Datatypes.RegisterDatatype(_eTcVnRotationAngle);
Datatypes.RegisterDatatype(_eTcVnRTrees);
Datatypes.RegisterDatatype(_eTcVnSignedNormalization);
Datatypes.RegisterDatatype(_eTcVnSolvePnPMethod);
Datatypes.RegisterDatatype(_eTcVnSta);
Datatypes.RegisterDatatype(_eTcVnStructuringElementShape);
Datatypes.RegisterDatatype(_eTcVnSvm);
Datatypes.RegisterDatatype(_eTcVnSvmKernelType);
Datatypes.RegisterDatatype(_eTcVnSvmSgdClassifierMarginType);
Datatypes.RegisterDatatype(_eTcVnSvmSgdClassifierType);
Datatypes.RegisterDatatype(_eTcVnTemplateMatchMethod);
Datatypes.RegisterDatatype(_eTcVnThresholdType);
Datatypes.RegisterDatatype(_eTcVnTimestamp);
Datatypes.RegisterDatatype(_eTcVnVectorCompareMethod);
Datatypes.RegisterDatatype(_eTcVnWorldCoordinateSystem);
Datatypes.RegisterDatatype(_eTcWatchdogAccumulationType);
Datatypes.RegisterDatatype(_gEV_CAMERA_STATE);
Datatypes.RegisterDatatype(_eTcVnDataLayout);
Datatypes.RegisterDatatype(_eTcVnReduceType);
Datatypes.RegisterDatatype(_eTcVnCircularityCalculationMethod);
Datatypes.RegisterDatatype(_eTcVnDataMatrixOptions);
Datatypes.RegisterDatatype(_eTcVnLayerNameType);
    
Datatypes.RegisterDatatype(_eTcVnComparisonOperator);
Datatypes.RegisterDatatype(_eTcVnDetectBarcodesWalshOptions);
Datatypes.RegisterDatatype(_eTcVnDetectPatternPointsOptions);
Datatypes.RegisterDatatype(_eTcVnDotCodeOptions);
Datatypes.RegisterDatatype(_eTcVnEdgeSelection);
Datatypes.RegisterDatatype(_eTcVnFindRoisMethod);
Datatypes.RegisterDatatype(_eTcVnJpegSampling);
Datatypes.RegisterDatatype(_eTcVnMergeRegionsOptions);
Datatypes.RegisterDatatype(_eTcVnPolarizedImageInterpolation);
Datatypes.RegisterDatatype(_eTcVnSalientFeaturesMethod);
// structs
Datatypes.RegisterDatatype(_gVSP_IMAGE_INFO);
Datatypes.RegisterDatatype(_gVSP_LEADER_PAYLOAD_IMAGE);
Datatypes.RegisterDatatype(_gVSP_PIXEL_FORMAT);
Datatypes.RegisterDatatype(_tcVnCameraCalibrationOptions);
Datatypes.RegisterDatatype(_tcVnCircularArc);
Datatypes.RegisterDatatype(_tcVnCodeGrades1D);
Datatypes.RegisterDatatype(_tcVnCodeGradesDM);
Datatypes.RegisterDatatype(_tcVnCodeGradesQR);
Datatypes.RegisterDatatype(_tcVnDMatch);
Datatypes.RegisterDatatype(_tcVnImageInfo);
Datatypes.RegisterDatatype(_tcVnKeyPoint);
//Datatypes.RegisterDatatype(_tcVnMatrix);
Datatypes.RegisterDatatype(_tcVnMoments);
Datatypes.RegisterDatatype(_tcVnParamsAGAST);
Datatypes.RegisterDatatype(_tcVnParamsAKAZE);
Datatypes.RegisterDatatype(_tcVnParamsBlobDetection);
Datatypes.RegisterDatatype(_tcVnParamsBRISK);
Datatypes.RegisterDatatype(_tcVnParamsFAST);
Datatypes.RegisterDatatype(_tcVnParamsGFTT);
Datatypes.RegisterDatatype(_tcVnParamsKAZE);
Datatypes.RegisterDatatype(_tcVnParamsMSER);
Datatypes.RegisterDatatype(_tcVnParamsORB);
Datatypes.RegisterDatatype(_tcVnParamsSB);
Datatypes.RegisterDatatype(_tcVnPixelFormat);
Datatypes.RegisterDatatype(_tcVnRectangle_DINT);
Datatypes.RegisterDatatype(_tcVnRectangle_UDINT);
Datatypes.RegisterDatatype(_tcVnRotatedRectangle);
Datatypes.RegisterDatatype(_tcVnSize2_REAL);

Datatypes.RegisterDatatype(_gVCP_ADDRESS_VALUE_PAIR);
Datatypes.RegisterDatatype(_tcVnSize2_DINT);
Datatypes.RegisterDatatype(_tcVnParamsFindRois);
Datatypes.RegisterDatatype(_tcVnParamsWalshBarcodeDetection);
// interfaces
Datatypes.RegisterDatatype(_iTcVnImage);
Datatypes.RegisterDatatype(_iTcVnContainer);
Datatypes.RegisterDatatype(_iTcVnDisplayableImage);
END_METHOD

END_FUNCTION_BLOCK

// Extensions/PreExecutionCheck/Alarms/PreExecutionCheckFailedAlarm
{attribute 'linkalways'} 
{attribute 'no_explicit_call' := 'This FB is a CLASS and must be accessed using methods or properties'}
{attribute 'enable_dynamic_creation'}
FUNCTION_BLOCK PUBLIC PreExecutionCheckFailedAlarm EXTENDS Alarm
VAR
	state : (CLEARED, RAISED);
	_reason : T_MAXSTRING;
END_VAR

PROPERTY Active : BOOL
GET
Active := state <> CLEARED;
END_GET
END_PROPERTY

METHOD PUBLIC Clear
_reason := '';
state := CLEARED;
END_METHOD

PROPERTY PUBLIC Message : T_MaxString
GET
Message := 'Pre-execution check failed';
END_GET
END_PROPERTY

METHOD PUBLIC Raise
VAR_INPUT
	Reason : T_MAXSTRING;
END_VAR
_reason := Reason;
state := RAISED;
END_METHOD

PROPERTY Reason : T_MaxString
GET
Reason := _reason;
END_GET
END_PROPERTY

END_FUNCTION_BLOCK

// Extensions/PreExecutionCheck/Checks/I_PreExecutionChecks
INTERFACE I_PreExecutionChecks

METHOD PUBLIC Fail
VAR_INPUT
	Message : T_MAXSTRING;
END_VAR
END_METHOD

PROPERTY PUBLIC Failed : BOOL
GET
END_GET
END_PROPERTY

METHOD PUBLIC IsFalse
VAR_INPUT
	Actual : BOOL;
	Message : T_MAXSTRING;
END_VAR
END_METHOD

METHOD PUBLIC IsTrue
VAR_INPUT
	Actual : BOOL;
	Message : T_MAXSTRING;
END_VAR
END_METHOD

END_INTERFACE

// Extensions/PreExecutionCheck/Checks/PreExecutionChecks
FUNCTION_BLOCK PreExecutionChecks IMPLEMENTS I_PreExecutionChecks
VAR
	hasFailed : BOOL;
	hasFailedReason : T_MAXSTRING;
END_VAR;

METHOD PUBLIC Fail
VAR_INPUT
	Message : T_MAXSTRING;
END_VAR
IF hasFailed THEN
	RETURN;
END_IF

hasFailed := TRUE;
hasFailedReason := Message;
END_METHOD

PROPERTY PUBLIC Failed : BOOL
GET
Failed := hasFailed;
END_GET
END_PROPERTY

METHOD PUBLIC IsFalse
VAR_INPUT
	Actual : BOOL;
	Message : T_MAXSTRING;
END_VAR
IF hasFailed THEN
	RETURN;
END_IF

IF NOT Actual THEN
	RETURN;
END_IF

hasFailed := TRUE;
hasFailedReason := Message;
END_METHOD

METHOD PUBLIC IsTrue
VAR_INPUT
	Actual : BOOL;
	Message : T_MAXSTRING;
END_VAR
IF hasFailed THEN
	RETURN;
END_IF

IF Actual THEN
	RETURN;
END_IF

hasFailed := TRUE;
hasFailedReason := Message;
END_METHOD

PROPERTY PUBLIC Passed : BOOL
GET
Passed := not hasFailed;
END_GET
END_PROPERTY

PROPERTY PUBLIC Reason : T_MAXSTRING
GET
Reason := hasFailedReason;
END_GET
END_PROPERTY

METHOD PUBLIC Reset
VAR_INPUT
END_VAR
hasFailed := FALSE;
hasFailedReason := '';
END_METHOD

END_FUNCTION_BLOCK

// Extensions/PreExecutionCheck/Interfaces/I_PreCheckedNode
INTERFACE I_PreCheckedNode EXTENDS I_Node

METHOD PreExecutionCheck
VAR_INPUT
	Check : I_PreExecutionChecks;
END_VAR
END_METHOD

END_INTERFACE

// Extensions/PreExecutionCheck/PreExecutionCheckExtension
FUNCTION_BLOCK PreExecutionCheckExtension EXTENDS Extension
VAR
	parentAsPreCheckedNode : I_PreCheckedNode;
	preExecutionCheckFailedAlarm : PreExecutionCheckFailedAlarm(THIS^);
	enable : _BOOL(TRUE);
END_VAR

METHOD FB_init : BOOL
VAR_INPUT
	bInitRetains : BOOL; // if TRUE, the retain variables are initialized (warm start / cold start)
	bInCopyCode : BOOL;  // if TRUE, the instance afterwards gets moved into the copy code (online change)
	Name : T_MAXSTRING;
	Parent : I_HostExtensions;
END_VAR
AddParameter('enable', enable);

IF NOT __QUERYINTERFACE(Parent, parentAsPreCheckedNode) THEN
	RETURN;
END_IF
END_METHOD

METHOD PUBLIC Check : BOOL
VAR_INPUT
END_VAR
VAR
	preExecutionChecks : PreExecutionChecks;
END_VAR
IF NOT enable.Value THEN
	IF preExecutionCheckFailedAlarm.Active THEN
		preExecutionCheckFailedAlarm.Clear();
	END_IF
	Check := TRUE;
	RETURN;
END_IF

parentAsPreCheckedNode.PreExecutionCheck(preExecutionChecks);
IF preExecutionChecks.Failed THEN
	preExecutionCheckFailedAlarm.Raise(preExecutionChecks.Reason);
	RETURN;
END_IF

preExecutionCheckFailedAlarm.Clear();
Check := TRUE;
END_METHOD

END_FUNCTION_BLOCK

// Extensions/WatchdogCheck/WatchdogCheckExtension
FUNCTION_BLOCK WatchdogCheckExtension EXTENDS Extension
VAR
	watchdogAlarm : FunctionFailedAlarm(THIS^);
	watchdogTimeInUs : _DINT(500000); // default
	hResult : HRESULT;
END_VAR

METHOD FB_init : BOOL
VAR_INPUT
	bInitRetains : BOOL; // if TRUE, the retain variables are initialized (warm start / cold start)
	bInCopyCode : BOOL;  // if TRUE, the instance afterwards gets moved into the copy code (online change)
	Name : T_MAXSTRING;
	Parent : I_HostExtensions;
END_VAR
AddParameter('watchdogTimeInUs', watchdogTimeInUs);
END_METHOD

METHOD PUBLIC Start
VAR_INPUT
END_VAR
watchdogAlarm.Clear();

IF watchdogTimeInUs.Value = 0 THEN
	RETURN;
END_IF

hResult := F_VN_StartRelWatchdog(watchdogTimeInUs.Value, S_OK);
END_METHOD

METHOD PUBLIC Stop
VAR_INPUT
END_VAR
hresult := F_VN_StopWatchdog(
	hrStartWatchdog := hresult);

IF FAILED(hresult) THEN
	watchdogAlarm.Raise('Watchdog', hresult);
END_IF
END_METHOD

END_FUNCTION_BLOCK

// Functions/Checks/ContainersHaveMatchingNumberOfElements
FUNCTION ContainersHaveMatchingNumberOfElements : BOOL
VAR_INPUT
	Container1 : ITcVnContainer;
	Container2 : ITcVnContainer;
END_VAR
VAR
    elementNum1 : ULINT;
    elementNum2 : ULINT;
END_VAR

IF NOT IsValidContainer(Container1) THEN
	RETURN;
END_IF

IF NOT IsValidContainer(Container2) THEN
	RETURN;
END_IF

IF NOT SUCCEEDED(Container1.GetElementNum(elementNum1)) THEN
    RETURN;
END_IF

IF NOT SUCCEEDED(Container2.GetElementNum(elementNum2)) THEN
    RETURN;
END_IF

ContainersHaveMatchingNumberOfElements := (elementNum1 = elementNum2);

END_FUNCTION

// Functions/Checks/IsValidContainer
FUNCTION IsValidContainer : BOOL
VAR_INPUT
    Container : ITcVnContainer;
END_VAR

IsValidContainer := Container <> 0;

END_FUNCTION

// Functions/Checks/ContainersHaveMatchingTypes
FUNCTION ContainersHaveMatchingTypes : BOOL
VAR_INPUT
	Container1 : ITcVnContainer;
	Container2 : ITcVnContainer;
END_VAR
VAR
    guid1 : GUID;
    guid2 : GUID;
END_VAR

IF NOT IsValidContainer(Container1) THEN
	RETURN;
END_IF

IF NOT IsValidContainer(Container2) THEN
	RETURN;
END_IF

IF NOT SUCCEEDED(Container1.GetTypeGuid(guid1)) THEN
    RETURN;
END_IF

IF NOT SUCCEEDED(Container2.GetTypeGuid(guid2)) THEN
    RETURN;
END_IF

ContainersHaveMatchingTypes := GuidsEqualByVal(guid1, guid2);

END_FUNCTION

// Functions/Checks/ImageHasCompatibleElementType
FUNCTION ImageHasCompatibleElementType : BOOL
VAR_INPUT
	Image : ITcVnImage;	
END_VAR
VAR_IN_OUT
	CompatibleElementTypes : ARRAY[*] OF ETcVnElementType;
END_VAR
VAR
	i : DINT;
END_VAR

IF NOT IsValidImage(Image) THEN
	RETURN;
END_IF

FOR i := LOWER_BOUND(CompatibleElementTypes, 1) TO UPPER_BOUND(CompatibleElementTypes, 1) DO
	IF ImageHasElementType(Image, CompatibleElementTypes[i]) THEN
		ImageHasCompatibleElementType := TRUE;
		RETURN;
	END_IF
END_FOR

END_FUNCTION

// Functions/Checks/IsValidImage
FUNCTION IsValidImage : BOOL
VAR_INPUT
    Image : ITcVnImage;
END_VAR

IsValidImage := Image <> 0;

END_FUNCTION

// Functions/Checks/ImageHasElementType
FUNCTION ImageHasElementType : BOOL
VAR_INPUT
	Image : ITcVnImage;
	ElementType : ETcVnElementType;
END_VAR

IF NOT IsValidImage(Image) THEN
	RETURN;
END_IF

ImageHasElementType := (ElementType = GetETcVnElementTypeFromImage(Image));

END_FUNCTION

// Functions/Helpers/GetETcVnElementTypeFromImage
FUNCTION GetETcVnElementTypeFromImage : ETcVnElementType
VAR_INPUT
	sourceImage : ITcVnImage;
END_VAR
VAR
	pixelFormat : TcVnPixelFormat;
END_VAR

IF NOT IsValidImage(sourceImage) THEN
	RETURN;
END_IF

sourceImage.GetPixelFormat(pixelFormat);

IF pixelFormat.nElementSize = 8 AND NOT pixelFormat.bSigned THEN
	GetETcVnElementTypeFromImage := ETcVnElementType.TCVN_ET_USINT;
ELSIF pixelFormat.nElementSize = 8 AND pixelFormat.bSigned THEN
	GetETcVnElementTypeFromImage := ETcVnElementType.TCVN_ET_SINT;
ELSIF pixelFormat.nElementSize = 16 AND NOT pixelFormat.bSigned THEN
	GetETcVnElementTypeFromImage := ETcVnElementType.TCVN_ET_UINT;
ELSIF pixelFormat.nElementSize = 16 AND pixelFormat.bSigned THEN
	GetETcVnElementTypeFromImage := ETcVnElementType.TCVN_ET_INT;
ELSIF pixelFormat.nElementSize = 32 AND NOT pixelFormat.bFloat THEN
	GetETcVnElementTypeFromImage := ETcVnElementType.TCVN_ET_DINT;
ELSIF pixelFormat.nElementSize = 32 AND pixelFormat.bFloat THEN
	GetETcVnElementTypeFromImage := ETcVnElementType.TCVN_ET_REAL;
ELSIF pixelFormat.nElementSize = 64 THEN
	GetETcVnElementTypeFromImage := ETcVnElementType.TCVN_ET_LREAL;
ELSE
	GetETcVnElementTypeFromImage := ETcVnElementType.TCVN_ET_SAME_AS_SOURCE;
END_IF

END_FUNCTION

// Functions/Checks/ImagesHaveMatchingChannels
FUNCTION ImagesHaveMatchingChannels : BOOL
VAR_INPUT
	Image1 : ITcVnImage;
	Image2 : ITcVnImage;
END_VAR
VAR
	pixelFormat1: TcVnPixelFormat;
	pixelFormat2: TcVnPixelFormat;
END_VAR

IF NOT IsValidImage(Image1) THEN
	RETURN;
END_IF

IF NOT IsValidImage(Image2) THEN
	RETURN;
END_IF

Image1.GetPixelFormat(pixelFormat1);
Image2.GetPixelFormat(pixelFormat2);

ImagesHaveMatchingChannels := (pixelFormat1.nChannels = pixelFormat2.nChannels);

END_FUNCTION

// Functions/Checks/ImagesHaveMatchingPixelFormats
FUNCTION ImagesHaveMatchingPixelFormats : BOOL
VAR_INPUT
	Image1 : ITcVnImage;
	Image2 : ITcVnImage;
END_VAR
VAR
	pixelFormat_1: TcVnPixelFormat;
	pixelFormat_2: TcVnPixelFormat;
	pointer_1 : POINTER TO BYTE;
	pointer_2 : POINTER TO BYTE;
END_VAR

IF NOT IsValidImage(Image1) THEN
	RETURN;
END_IF

IF NOT IsValidImage(Image2) THEN
	RETURN;
END_IF

Image1.GetPixelFormat(pixelFormat_1);
Image2.GetPixelFormat(pixelFormat_2);

pointer_1 := ADR(pixelFormat_1);
pointer_2 := ADR(pixelFormat_2);

ImagesHaveMatchingPixelFormats := (MEMCMP(pointer_1, pointer_2, SIZEOF(pixelFormat_1)) = 0);

END_FUNCTION

// Functions/Checks/IsImage1SizeEqualToImage2Size
FUNCTION IsImage1SizeEqualToImage2Size : BOOL
VAR_INPUT
    Image1 : ITcVnImage;
    Image2 : ITcVnImage;
END_VAR
VAR
    image1Width : UDINT;
    image1Height : UDINT;
    image2Width : UDINT;
    image2Height : UDINT;
END_VAR

IF NOT IsValidImage(Image1) THEN
    RETURN;
END_IF

IF NOT IsValidImage(Image2) THEN
    RETURN;
END_IF

Image1.GetWidth(image1Width);
Image1.GetHeight(image1Height);

Image2.GetWidth(image2Width);
Image2.GetHeight(image2Height);

IF (image1Width <> image2Width) OR_ELSE (image1Height <> image2Height) THEN
    RETURN;
END_IF

IsImage1SizeEqualToImage2Size := TRUE;

END_FUNCTION

// Functions/Checks/IsImage1WidthEqualToImage2Width
FUNCTION IsImage1WidthEqualToImage2Width : BOOL
VAR_INPUT
    Image1 : ITcVnImage;
    Image2 : ITcVnImage;
END_VAR
VAR
    image1Width : UDINT;
    image2Width : UDINT;
END_VAR

IF NOT IsValidImage(Image1) THEN
    RETURN;
END_IF

IF NOT IsValidImage(Image2) THEN
    RETURN;
END_IF

Image1.GetWidth(image1Width);
Image2.GetWidth(image2Width);

IF (image1Width <> image2Width) THEN
    RETURN;
END_IF

IsImage1WidthEqualToImage2Width := TRUE;

END_FUNCTION

// Functions/Checks/IsMaxValueCompatibleWithPixelDepth
FUNCTION IsMaxValueCompatibleWithPixelDepth : BOOL
VAR_INPUT
    Value : LREAL;
    PixelDepth : UINT;
END_VAR
VAR
    minimumAllowedValue : LREAL;
    maximumAllowedValue : LREAL;
END_VAR

CASE PixelDepth OF
    8:
        minimumAllowedValue := 0.0;
        TryConvert_USINT_TO_LREAL(DatatypeLimits.USINT_MAX_VALUE, maximumAllowedValue);
    16:
        minimumAllowedValue := 0.0;
        TryConvert_UINT_TO_LREAL(DatatypeLimits.UINT_MAX_VALUE, maximumAllowedValue);
    32:
        TryConvert_REAL_TO_LREAL(DatatypeLimits.REAL_MIN_VALUE, minimumAllowedValue);
        TryConvert_REAL_TO_LREAL(DatatypeLimits.REAL_MAX_VALUE, maximumAllowedValue);
    64:
        minimumAllowedValue := DatatypeLimits.LREAL_MIN_VALUE;
        maximumAllowedValue := DatatypeLimits.LREAL_MAX_VALUE;
ELSE
    ;
END_CASE

IF (Value < minimumAllowedValue) OR (Value > maximumAllowedValue) THEN
    RETURN;
END_IF

IsMaxValueCompatibleWithPixelDepth := TRUE;

END_FUNCTION

// Functions/Checks/IsRemapMapPairValid
FUNCTION IsRemapMapPairValid : BOOL
VAR_INPUT
    Map1 : ITcVnImage;
    Map2 : ITcVnImage;
END_VAR
VAR
    format1 : TcVnPixelFormat;
    format2 : TcVnPixelFormat;
    map1IsReal : BOOL;
    map1IsInt : BOOL;
END_VAR

// The map pair determines the destination size; it need not match the source image size.
IF NOT IsValidImage(Map1) THEN
    RETURN;
END_IF
IF FAILED(Map1.GetPixelFormat(format1)) THEN
    RETURN;
END_IF
map1IsReal := ImageHasElementType(Map1, ETcVnElementType.TCVN_ET_REAL);
map1IsInt := ImageHasElementType(Map1, ETcVnElementType.TCVN_ET_INT);

IF Map2 = 0 THEN
    // Interleaved floating-point coordinates, or rounded fixed-point coordinates.
    IsRemapMapPairValid := (format1.nChannels = 2) AND (map1IsReal OR map1IsInt);
    RETURN;
END_IF
IF FAILED(Map2.GetPixelFormat(format2)) THEN
    RETURN;
END_IF
IF NOT IsImage1SizeEqualToImage2Size(Map1, Map2) THEN
    RETURN;
END_IF
IF format2.nChannels <> 1 THEN
    RETURN;
END_IF
// Separate floating-point X/Y maps, or fixed-point coordinates plus interpolation coefficients.
IsRemapMapPairValid := ((format1.nChannels = 1) AND map1IsReal AND
                       ImageHasElementType(Map2, ETcVnElementType.TCVN_ET_REAL)) OR
                      ((format1.nChannels = 2) AND map1IsInt AND
                       ImageHasElementType(Map2, ETcVnElementType.TCVN_ET_UINT));

END_FUNCTION

// Functions/Checks/IsRoiSizeOK_Dint
FUNCTION IsRoiSizeOK_Dint : BOOL
VAR_INPUT
    RoiRectangle : TcVnRectangle_DINT;
    ImageWidth : UDINT;
    ImageHeight : UDINT;
END_VAR
VAR
    width : DINT;
    height : DINT;
END_VAR

IF NOT TryConvert_UDINT_TO_DINT(ImageWidth, width) THEN
    RETURN;
END_IF

IF NOT TryConvert_UDINT_TO_DINT(ImageHeight, height) THEN
    RETURN;
END_IF

IF NOT (RoiRectangle.nX < width) THEN
	RETURN;
END_IF

IF NOT (RoiRectangle.nY < height) THEN
	RETURN;
END_IF

IF NOT (RoiRectangle.nWidth <= (width - RoiRectangle.nX)) THEN
	RETURN;
END_IF

IF NOT (RoiRectangle.nHeight <= (height - RoiRectangle.nY)) THEN
	RETURN;
END_IF

IsRoiSizeOK_Dint := TRUE;

END_FUNCTION

// Functions/Checks/IsRoiSizeOK_Udint
FUNCTION IsRoiSizeOK_Udint : BOOL
VAR_INPUT
    RoiRectangle : TcVnRectangle_UDINT;
    ImageWidth : UDINT;
    ImageHeight : UDINT;
END_VAR

IF NOT (RoiRectangle.nX < ImageWidth) THEN
	RETURN;
END_IF

IF NOT (RoiRectangle.nY < ImageHeight) THEN
	RETURN;
END_IF

IF NOT (RoiRectangle.nWidth <= (ImageWidth - RoiRectangle.nX)) THEN
	RETURN;
END_IF

IF NOT (RoiRectangle.nHeight <= (ImageHeight - RoiRectangle.nY)) THEN
	RETURN;
END_IF

IsRoiSizeOK_Udint := TRUE;

END_FUNCTION

// Functions/Checks/IsTemplateImageSmallerThanSourceImage
FUNCTION IsTemplateImageSmallerThanSourceImage : BOOL
VAR_INPUT
    SourceImage : ITcVnImage;
    TemplateImage : ITcVnImage;
END_VAR
VAR
    sourceWidth : UDINT;
    sourceHeight : UDINT;
    templateWidth : UDINT;
    templateHeight : UDINT;
END_VAR

IF NOT IsValidImage(SourceImage) THEN
    RETURN;
END_IF

IF NOT IsValidImage(TemplateImage) THEN
    RETURN;
END_IF

SourceImage.GetWidth(sourceWidth);
SourceImage.GetHeight(sourceHeight);
TemplateImage.GetWidth(templateWidth);
TemplateImage.GetHeight(templateHeight);

IF (templateWidth >= sourceWidth) THEN
    RETURN;
END_IF

IF (templateHeight >= sourceHeight) THEN
    RETURN;
END_IF

IsTemplateImageSmallerThanSourceImage := TRUE;

END_FUNCTION

// Functions/Checks/IsValidIterator
FUNCTION IsValidIterator : BOOL
VAR_INPUT
    Iterator : ITcVnIteratorBase;
END_VAR

IsValidIterator := Iterator <> 0;

END_FUNCTION

// Nodes/Algebraic Container Ops/AddTo/Node_F_VN_AddToContainerElements_DINT
{attribute 'linkalways'} 
{attribute 'no_explicit_call' := 'This FB is a CLASS and must be accessed using methods or properties'}
{attribute 'enable_dynamic_creation'}
FUNCTION_BLOCK Node_F_VN_AddToContainerElements_DINT EXTENDS VisionNode
VAR
    nValue : _DINT(0);
    ipContainer : _ITcVnContainer;
    hrPrev : _HRESULT(S_OK);
    hresult : _HRESULT(S_OK);
END_VAR

METHOD FB_init : BOOL
VAR_INPUT
    bInitRetains : BOOL; // if TRUE, the retain variables are initialized (warm start / cold start)
    bInCopyCode : BOOL;  // if TRUE, the instance afterwards gets moved into the copy code (online change)
END_VAR
AddParameter('nValue', nValue);
AddInput('ipContainer', ipContainer);
AddInput('hrPrev', hrPrev);
AddOutput('ipContainer', ipContainer);
AddOutput('hresult',hresult);
END_METHOD

METHOD PUBLIC  Clone : I_Node
VAR
    pNode : POINTER TO Node_F_VN_AddToContainerElements_DINT;
END_VAR
pNode := __NEW(Node_F_VN_AddToContainerElements_DINT);
Clone := pNode^;
END_METHOD

METHOD PROTECTED OnExecute
hresult.Value := F_VN_AddToContainerElements_DINT(
    nValue := nValue.Value,
    ipContainer := ipContainer.Value,
    hrPrev:= hrPrev.Value);
END_METHOD

METHOD PUBLIC PreExecutionCheck
VAR_INPUT
    Check : I_PreExecutionChecks;
END_VAR
Check.IsTrue(ipContainer.IsValid, 'ipContainer must be a valid container');
Check.IsTrue(ipContainer.IsType(TC_GLOBAL_CONST_LIST.ContainerType_Vector_DINT), 'ipContainer contains incorrect type');
END_METHOD

END_FUNCTION_BLOCK

// Nodes/VisionNode/VisionNode
FUNCTION_BLOCK ABSTRACT VisionNode EXTENDS Node IMPLEMENTS I_PreCheckedNode
VAR
	preExecutionCheckExtension : PreExecutionCheckExtension('precheck', THIS^);
	watchdogCheckExtension : WatchdogCheckExtension('watchdog', THIS^);
END_VAR

METHOD PUBLIC Execute
VAR
END_VAR
IF NOT preExecutionCheckExtension.Check() THEN
	RETURN;
END_IF

watchdogCheckExtension.Start();
SUPER^.Execute();
watchdogCheckExtension.Stop();
END_METHOD

METHOD PUBLIC ABSTRACT PreExecutionCheck
VAR_INPUT
	Check : I_PreExecutionChecks;
END_VAR
END_METHOD

END_FUNCTION_BLOCK

// Nodes/Algebraic Container Ops/AddTo/Node_F_VN_AddToContainerElements_INT
{attribute 'linkalways'} 
{attribute 'no_explicit_call' := 'This FB is a CLASS and must be accessed using methods or properties'}
{attribute 'enable_dynamic_creation'}
FUNCTION_BLOCK Node_F_VN_AddToContainerElements_INT EXTENDS VisionNode
VAR
    nValue : _INT(0);
    ipContainer : _ITcVnContainer;
    hrPrev : _HRESULT(S_OK);
    hresult : _HRESULT(S_OK);
END_VAR

METHOD FB_init : BOOL
VAR_INPUT
    bInitRetains : BOOL; // if TRUE, the retain variables are initialized (warm start / cold start)
    bInCopyCode : BOOL;  // if TRUE, the instance afterwards gets moved into the copy code (online change)
END_VAR
AddParameter('nValue', nValue);
AddInput('ipContainer', ipContainer);
AddInput('hrPrev', hrPrev);
AddOutput('ipContainer', ipContainer);
AddOutput('hresult',hresult);
END_METHOD

METHOD PUBLIC  Clone : I_Node
VAR
    pNode : POINTER TO Node_F_VN_AddToContainerElements_INT;
END_VAR
pNode := __NEW(Node_F_VN_AddToContainerElements_INT);
Clone := pNode^;
END_METHOD

METHOD PROTECTED OnExecute
hresult.Value := F_VN_AddToContainerElements_INT(
    nValue := nValue.Value,
    ipContainer := ipContainer.Value,
    hrPrev:= hrPrev.Value);
END_METHOD

METHOD PUBLIC PreExecutionCheck
VAR_INPUT
    Check : I_PreExecutionChecks;
END_VAR
Check.IsTrue(ipContainer.IsValid, 'ipContainer must be a valid container');
Check.IsTrue(ipContainer.IsType(TC_GLOBAL_CONST_LIST.ContainerType_Vector_INT), 'ipContainer contains incorrect type');
END_METHOD

END_FUNCTION_BLOCK

// Nodes/Algebraic Container Ops/AddTo/Node_F_VN_AddToContainerElements_LREAL
{attribute 'linkalways'} 
{attribute 'no_explicit_call' := 'This FB is a CLASS and must be accessed using methods or properties'}
{attribute 'enable_dynamic_creation'}
FUNCTION_BLOCK Node_F_VN_AddToContainerElements_LREAL EXTENDS VisionNode
VAR
    fValue : _LREAL(0.0);
    ipContainer : _ITcVnContainer;
    hrPrev : _HRESULT(S_OK);
    hresult : _HRESULT(S_OK);
END_VAR

METHOD FB_init : BOOL
VAR_INPUT
    bInitRetains : BOOL; // if TRUE, the retain variables are initialized (warm start / cold start)
    bInCopyCode : BOOL;  // if TRUE, the instance afterwards gets moved into the copy code (online change)
END_VAR
AddParameter('fValue', fValue);
AddInput('ipContainer', ipContainer);
AddInput('hrPrev', hrPrev);
AddOutput('ipContainer', ipContainer);
AddOutput('hresult',hresult);
END_METHOD

METHOD PUBLIC  Clone : I_Node
VAR
    pNode : POINTER TO Node_F_VN_AddToContainerElements_LREAL;
END_VAR
pNode := __NEW(Node_F_VN_AddToContainerElements_LREAL);
Clone := pNode^;
END_METHOD

METHOD PROTECTED OnExecute
hresult.Value := F_VN_AddToContainerElements_LREAL(
    fValue := fValue.Value,
    ipContainer := ipContainer.Value,
    hrPrev:= hrPrev.Value);
END_METHOD

METHOD PUBLIC PreExecutionCheck
VAR_INPUT
    Check : I_PreExecutionChecks;
END_VAR
Check.IsTrue(ipContainer.IsValid, 'ipContainer must be a valid container');
Check.IsTrue(ipContainer.IsType(TC_GLOBAL_CONST_LIST.ContainerType_Vector_LREAL), 'ipContainer contains incorrect type');
END_METHOD

END_FUNCTION_BLOCK

// Nodes/Algebraic Container Ops/AddTo/Node_F_VN_AddToContainerElements_REAL
{attribute 'linkalways'} 
{attribute 'no_explicit_call' := 'This FB is a CLASS and must be accessed using methods or properties'}
{attribute 'enable_dynamic_creation'}
FUNCTION_BLOCK Node_F_VN_AddToContainerElements_REAL EXTENDS VisionNode
VAR
    fValue : _REAL(0.0);
    ipContainer : _ITcVnContainer;
    hrPrev : _HRESULT(S_OK);
    hresult : _HRESULT(S_OK);
END_VAR

METHOD FB_init : BOOL
VAR_INPUT
    bInitRetains : BOOL; // if TRUE, the retain variables are initialized (warm start / cold start)
    bInCopyCode : BOOL;  // if TRUE, the instance afterwards gets moved into the copy code (online change)
END_VAR
AddParameter('fValue', fValue);
AddInput('ipContainer', ipContainer);
AddInput('hrPrev', hrPrev);
AddOutput('ipContainer', ipContainer);
AddOutput('hresult',hresult);
END_METHOD

METHOD PUBLIC  Clone : I_Node
VAR
    pNode : POINTER TO Node_F_VN_AddToContainerElements_REAL;
END_VAR
pNode := __NEW(Node_F_VN_AddToContainerElements_REAL);
Clone := pNode^;
END_METHOD

METHOD PROTECTED OnExecute
hresult.Value := F_VN_AddToContainerElements_REAL(
    fValue := fValue.Value,
    ipContainer := ipContainer.Value,
    hrPrev:= hrPrev.Value);
END_METHOD

METHOD PUBLIC PreExecutionCheck
VAR_INPUT
    Check : I_PreExecutionChecks;
END_VAR
Check.IsTrue(ipContainer.IsValid, 'ipContainer must be a valid container');
Check.IsTrue(ipContainer.IsType(TC_GLOBAL_CONST_LIST.ContainerType_Vector_REAL), 'ipContainer contains incorrect type');
END_METHOD

END_FUNCTION_BLOCK

// Nodes/Algebraic Container Ops/AddTo/Node_F_VN_AddToContainerElements_SINT
{attribute 'linkalways'} 
{attribute 'no_explicit_call' := 'This FB is a CLASS and must be accessed using methods or properties'}
{attribute 'enable_dynamic_creation'}
FUNCTION_BLOCK Node_F_VN_AddToContainerElements_SINT EXTENDS VisionNode
VAR
    nValue : _SINT(0);
    ipContainer : _ITcVnContainer;
    hrPrev : _HRESULT(S_OK);
    hresult : _HRESULT(S_OK);
END_VAR

METHOD FB_init : BOOL
VAR_INPUT
    bInitRetains : BOOL; // if TRUE, the retain variables are initialized (warm start / cold start)
    bInCopyCode : BOOL;  // if TRUE, the instance afterwards gets moved into the copy code (online change)
END_VAR
AddParameter('nValue', nValue);
AddInput('ipContainer', ipContainer);
AddInput('hrPrev', hrPrev);
AddOutput('ipContainer', ipContainer);
AddOutput('hresult',hresult);
END_METHOD

METHOD PUBLIC  Clone : I_Node
VAR
    pNode : POINTER TO Node_F_VN_AddToContainerElements_SINT;
END_VAR
pNode := __NEW(Node_F_VN_AddToContainerElements_SINT);
Clone := pNode^;
END_METHOD

METHOD PROTECTED OnExecute
hresult.Value := F_VN_AddToContainerElements_SINT(
    nValue := nValue.Value,
    ipContainer := ipContainer.Value,
    hrPrev:= hrPrev.Value);
END_METHOD

METHOD PUBLIC PreExecutionCheck
VAR_INPUT
    Check : I_PreExecutionChecks;
END_VAR
Check.IsTrue(ipContainer.IsValid, 'ipContainer must be a valid container');
Check.IsTrue(ipContainer.IsType(TC_GLOBAL_CONST_LIST.ContainerType_Vector_SINT), 'ipContainer contains incorrect type');
END_METHOD

END_FUNCTION_BLOCK

// Nodes/Algebraic Container Ops/AddTo/Node_F_VN_AddToContainerElements_TcVnKeyPoint
{attribute 'linkalways'} 
{attribute 'no_explicit_call' := 'This FB is a CLASS and must be accessed using methods or properties'}
{attribute 'enable_dynamic_creation'}
FUNCTION_BLOCK Node_F_VN_AddToContainerElements_TcVnKeyPoint EXTENDS VisionNode
VAR
    stValue : _TcVnKeyPoint;
    ipContainer : _ITcVnContainer;
    hrPrev : _HRESULT(S_OK);
    hresult : _HRESULT(S_OK);
END_VAR

METHOD FB_init : BOOL
VAR_INPUT
    bInitRetains : BOOL; // if TRUE, the retain variables are initialized (warm start / cold start)
    bInCopyCode : BOOL;  // if TRUE, the instance afterwards gets moved into the copy code (online change)
END_VAR
AddInput('stValue', stValue);
AddInput('ipContainer', ipContainer);
AddInput('hrPrev', hrPrev);
AddOutput('ipContainer', ipContainer);
AddOutput('hresult',hresult);
END_METHOD

METHOD PUBLIC  Clone : I_Node
VAR
    pNode : POINTER TO Node_F_VN_AddToContainerElements_TcVnKeyPoint;
END_VAR
pNode := __NEW(Node_F_VN_AddToContainerElements_TcVnKeyPoint);
Clone := pNode^;
END_METHOD

METHOD PROTECTED OnExecute
hresult.Value := F_VN_AddToContainerElements_TcVnKeyPoint(
    stValue := stValue.Value,
    ipContainer := ipContainer.Value,
    hrPrev:= hrPrev.Value);
END_METHOD

METHOD PUBLIC PreExecutionCheck
VAR_INPUT
    Check : I_PreExecutionChecks;
END_VAR
Check.IsTrue(ipContainer.IsValid, 'ipContainer must be a valid container');
Check.IsTrue(ipContainer.IsType(TC_GLOBAL_CONST_LIST.ContainerType_Vector_TcVnKeyPoint), 'ipContainer contains incorrect type');
END_METHOD

END_FUNCTION_BLOCK

// Nodes/Algebraic Container Ops/AddTo/Node_F_VN_AddToContainerElements_TcVnPoint2_DINT
{attribute 'linkalways'} 
{attribute 'no_explicit_call' := 'This FB is a CLASS and must be accessed using methods or properties'}
{attribute 'enable_dynamic_creation'}
FUNCTION_BLOCK Node_F_VN_AddToContainerElements_TcVnPoint2_DINT EXTENDS VisionNode
VAR
    aValue : _TcVnPoint2_DINT;
    ipContainer : _ITcVnContainer;
    hrPrev : _HRESULT(S_OK);
    hresult : _HRESULT(S_OK);
END_VAR

METHOD FB_init : BOOL
VAR_INPUT
    bInitRetains : BOOL; // if TRUE, the retain variables are initialized (warm start / cold start)
    bInCopyCode : BOOL;  // if TRUE, the instance afterwards gets moved into the copy code (online change)
END_VAR
AddInput('aValue', aValue);
AddInput('ipContainer', ipContainer);
AddInput('hrPrev', hrPrev);
AddOutput('ipContainer', ipContainer);
AddOutput('hresult',hresult);
END_METHOD

METHOD PUBLIC  Clone : I_Node
VAR
    pNode : POINTER TO Node_F_VN_AddToContainerElements_TcVnPoint2_DINT;
END_VAR
pNode := __NEW(Node_F_VN_AddToContainerElements_TcVnPoint2_DINT);
Clone := pNode^;
END_METHOD

METHOD PROTECTED OnExecute
hresult.Value := F_VN_AddToContainerElements_TcVnPoint2_DINT(
    aValue := aValue.Value,
    ipContainer := ipContainer.Value,
    hrPrev:= hrPrev.Value);
END_METHOD

METHOD PUBLIC PreExecutionCheck
VAR_INPUT
    Check : I_PreExecutionChecks;
END_VAR
Check.IsTrue(ipContainer.IsValid, 'ipContainer must be a valid container');
Check.IsTrue(ipContainer.IsType(TC_GLOBAL_CONST_LIST.ContainerType_Vector_TcVnPoint2_DINT), 'ipContainer contains incorrect type');
END_METHOD

END_FUNCTION_BLOCK

// Nodes/Algebraic Container Ops/AddTo/Node_F_VN_AddToContainerElements_TcVnPoint2_LREAL
{attribute 'linkalways'} 
{attribute 'no_explicit_call' := 'This FB is a CLASS and must be accessed using methods or properties'}
{attribute 'enable_dynamic_creation'}
FUNCTION_BLOCK Node_F_VN_AddToContainerElements_TcVnPoint2_LREAL EXTENDS VisionNode
VAR
    aValue : _TcVnPoint2_LREAL;
    ipContainer : _ITcVnContainer;
    hrPrev : _HRESULT(S_OK);
    hresult : _HRESULT(S_OK);
END_VAR

METHOD FB_init : BOOL
VAR_INPUT
    bInitRetains : BOOL; // if TRUE, the retain variables are initialized (warm start / cold start)
    bInCopyCode : BOOL;  // if TRUE, the instance afterwards gets moved into the copy code (online change)
END_VAR
AddInput('aValue', aValue);
AddInput('ipContainer', ipContainer);
AddInput('hrPrev', hrPrev);
AddOutput('ipContainer', ipContainer);
AddOutput('hresult',hresult);
END_METHOD

METHOD PUBLIC  Clone : I_Node
VAR
    pNode : POINTER TO Node_F_VN_AddToContainerElements_TcVnPoint2_LREAL;
END_VAR
pNode := __NEW(Node_F_VN_AddToContainerElements_TcVnPoint2_LREAL);
Clone := pNode^;
END_METHOD

METHOD PROTECTED OnExecute
hresult.Value := F_VN_AddToContainerElements_TcVnPoint2_LREAL(
    aValue := aValue.Value,
    ipContainer := ipContainer.Value,
    hrPrev:= hrPrev.Value);
END_METHOD

METHOD PUBLIC PreExecutionCheck
VAR_INPUT
    Check : I_PreExecutionChecks;
END_VAR
Check.IsTrue(ipContainer.IsValid, 'ipContainer must be a valid container');
Check.IsTrue(ipContainer.IsType(TC_GLOBAL_CONST_LIST.ContainerType_Vector_TcVnPoint2_LREAL), 'ipContainer contains incorrect type');
END_METHOD

END_FUNCTION_BLOCK

// Nodes/Algebraic Container Ops/AddTo/Node_F_VN_AddToContainerElements_TcVnPoint2_REAL
{attribute 'linkalways'} 
{attribute 'no_explicit_call' := 'This FB is a CLASS and must be accessed using methods or properties'}
{attribute 'enable_dynamic_creation'}
FUNCTION_BLOCK Node_F_VN_AddToContainerElements_TcVnPoint2_REAL EXTENDS VisionNode
VAR
    aValue : _TcVnPoint2_REAL;
    ipContainer : _ITcVnContainer;
    hrPrev : _HRESULT(S_OK);
    hresult : _HRESULT(S_OK);
END_VAR

METHOD FB_init : BOOL
VAR_INPUT
    bInitRetains : BOOL; // if TRUE, the retain variables are initialized (warm start / cold start)
    bInCopyCode : BOOL;  // if TRUE, the instance afterwards gets moved into the copy code (online change)
END_VAR
AddInput('aValue', aValue);
AddInput('ipContainer', ipContainer);
AddInput('hrPrev', hrPrev);
AddOutput('ipContainer', ipContainer);
AddOutput('hresult',hresult);
END_METHOD

METHOD PUBLIC  Clone : I_Node
VAR
    pNode : POINTER TO Node_F_VN_AddToContainerElements_TcVnPoint2_REAL;
END_VAR
pNode := __NEW(Node_F_VN_AddToContainerElements_TcVnPoint2_REAL);
Clone := pNode^;
END_METHOD

METHOD PROTECTED OnExecute
hresult.Value := F_VN_AddToContainerElements_TcVnPoint2_REAL(
    aValue := aValue.Value,
    ipContainer := ipContainer.Value,
    hrPrev:= hrPrev.Value);
END_METHOD

METHOD PUBLIC PreExecutionCheck
VAR_INPUT
    Check : I_PreExecutionChecks;
END_VAR
Check.IsTrue(ipContainer.IsValid, 'ipContainer must be a valid container');
Check.IsTrue(ipContainer.IsType(TC_GLOBAL_CONST_LIST.ContainerType_Vector_TcVnPoint2_REAL), 'ipContainer contains incorrect type');
END_METHOD

END_FUNCTION_BLOCK

// Nodes/Algebraic Container Ops/AddTo/Node_F_VN_AddToContainerElements_TcVnPoint3_LREAL
{attribute 'linkalways'} 
{attribute 'no_explicit_call' := 'This FB is a CLASS and must be accessed using methods or properties'}
{attribute 'enable_dynamic_creation'}
FUNCTION_BLOCK Node_F_VN_AddToContainerElements_TcVnPoint3_LREAL EXTENDS VisionNode
VAR
    aValue : _TcVnPoint3_LREAL;
    ipContainer : _ITcVnContainer;
    hrPrev : _HRESULT(S_OK);
    hresult : _HRESULT(S_OK);
END_VAR

METHOD FB_init : BOOL
VAR_INPUT
    bInitRetains : BOOL; // if TRUE, the retain variables are initialized (warm start / cold start)
    bInCopyCode : BOOL;  // if TRUE, the instance afterwards gets moved into the copy code (online change)
END_VAR
AddInput('aValue', aValue);
AddInput('ipContainer', ipContainer);
AddInput('hrPrev', hrPrev);
AddOutput('ipContainer', ipContainer);
AddOutput('hresult',hresult);
END_METHOD

METHOD PUBLIC  Clone : I_Node
VAR
    pNode : POINTER TO Node_F_VN_AddToContainerElements_TcVnPoint3_LREAL;
END_VAR
pNode := __NEW(Node_F_VN_AddToContainerElements_TcVnPoint3_LREAL);
Clone := pNode^;
END_METHOD

METHOD PROTECTED OnExecute
hresult.Value := F_VN_AddToContainerElements_TcVnPoint3_LREAL(
    aValue := aValue.Value,
    ipContainer := ipContainer.Value,
    hrPrev:= hrPrev.Value);
END_METHOD

METHOD PUBLIC PreExecutionCheck
VAR_INPUT
    Check : I_PreExecutionChecks;
END_VAR
Check.IsTrue(ipContainer.IsValid, 'ipContainer must be a valid container');
Check.IsTrue(ipContainer.IsType(TC_GLOBAL_CONST_LIST.ContainerType_Vector_TcVnPoint3_LREAL), 'ipContainer contains incorrect type');
END_METHOD

END_FUNCTION_BLOCK

// Nodes/Algebraic Container Ops/AddTo/Node_F_VN_AddToContainerElements_TcVnPoint3_REAL
{attribute 'linkalways'} 
{attribute 'no_explicit_call' := 'This FB is a CLASS and must be accessed using methods or properties'}
{attribute 'enable_dynamic_creation'}
FUNCTION_BLOCK Node_F_VN_AddToContainerElements_TcVnPoint3_REAL EXTENDS VisionNode
VAR
    aValue : _TcVnPoint3_REAL;
    ipContainer : _ITcVnContainer;
    hrPrev : _HRESULT(S_OK);
    hresult : _HRESULT(S_OK);
END_VAR

METHOD FB_init : BOOL
VAR_INPUT
    bInitRetains : BOOL; // if TRUE, the retain variables are initialized (warm start / cold start)
    bInCopyCode : BOOL;  // if TRUE, the instance afterwards gets moved into the copy code (online change)
END_VAR
AddInput('aValue', aValue);
AddInput('ipContainer', ipContainer);
AddInput('hrPrev', hrPrev);
AddOutput('ipContainer', ipContainer);
AddOutput('hresult',hresult);
END_METHOD

METHOD PUBLIC  Clone : I_Node
VAR
    pNode : POINTER TO Node_F_VN_AddToContainerElements_TcVnPoint3_REAL;
END_VAR
pNode := __NEW(Node_F_VN_AddToContainerElements_TcVnPoint3_REAL);
Clone := pNode^;
END_METHOD

METHOD PROTECTED OnExecute
hresult.Value := F_VN_AddToContainerElements_TcVnPoint3_REAL(
    aValue := aValue.Value,
    ipContainer := ipContainer.Value,
    hrPrev:= hrPrev.Value);
END_METHOD

METHOD PUBLIC PreExecutionCheck
VAR_INPUT
    Check : I_PreExecutionChecks;
END_VAR
Check.IsTrue(ipContainer.IsValid, 'ipContainer must be a valid container');
Check.IsTrue(ipContainer.IsType(TC_GLOBAL_CONST_LIST.ContainerType_Vector_TcVnPoint3_REAL), 'ipContainer contains incorrect type');
END_METHOD

END_FUNCTION_BLOCK

// Nodes/Algebraic Container Ops/AddTo/Node_F_VN_AddToContainerElements_TcVnRectangle_DINT
{attribute 'linkalways'} 
{attribute 'no_explicit_call' := 'This FB is a CLASS and must be accessed using methods or properties'}
{attribute 'enable_dynamic_creation'}
FUNCTION_BLOCK Node_F_VN_AddToContainerElements_TcVnRectangle_DINT EXTENDS VisionNode
VAR
    stValue : _TcVnRectangle_DINT;
    ipContainer : _ITcVnContainer;
    hrPrev : _HRESULT(S_OK);
    hresult : _HRESULT(S_OK);
END_VAR

METHOD FB_init : BOOL
VAR_INPUT
    bInitRetains : BOOL; // if TRUE, the retain variables are initialized (warm start / cold start)
    bInCopyCode : BOOL;  // if TRUE, the instance afterwards gets moved into the copy code (online change)
END_VAR
AddInput('stValue', stValue);
AddInput('ipContainer', ipContainer);
AddInput('hrPrev', hrPrev);
AddOutput('ipContainer', ipContainer);
AddOutput('hresult',hresult);
END_METHOD

METHOD PUBLIC  Clone : I_Node
VAR
    pNode : POINTER TO Node_F_VN_AddToContainerElements_TcVnRectangle_DINT;
END_VAR
pNode := __NEW(Node_F_VN_AddToContainerElements_TcVnRectangle_DINT);
Clone := pNode^;
END_METHOD

METHOD PROTECTED OnExecute
hresult.Value := F_VN_AddToContainerElements_TcVnRectangle_DINT(
    stValue := stValue.Value,
    ipContainer := ipContainer.Value,
    hrPrev:= hrPrev.Value);
END_METHOD

METHOD PUBLIC PreExecutionCheck
VAR_INPUT
    Check : I_PreExecutionChecks;
END_VAR
Check.IsTrue(ipContainer.IsValid, 'ipContainer must be a valid container');
Check.IsTrue(ipContainer.IsType(TC_GLOBAL_CONST_LIST.ContainerType_Vector_TcVnRectangle_DINT), 'ipContainer contains incorrect type');
END_METHOD

END_FUNCTION_BLOCK

// Nodes/Algebraic Container Ops/AddTo/Node_F_VN_AddToContainerElements_TcVnRotatedRectangle
{attribute 'linkalways'} 
{attribute 'no_explicit_call' := 'This FB is a CLASS and must be accessed using methods or properties'}
{attribute 'enable_dynamic_creation'}
FUNCTION_BLOCK Node_F_VN_AddToContainerElements_TcVnRotatedRectangle EXTENDS VisionNode
VAR
    stValue : _TcVnRotatedRectangle;
    ipContainer : _ITcVnContainer;
    hrPrev : _HRESULT(S_OK);
    hresult : _HRESULT(S_OK);
END_VAR

METHOD FB_init : BOOL
VAR_INPUT
    bInitRetains : BOOL; // if TRUE, the retain variables are initialized (warm start / cold start)
    bInCopyCode : BOOL;  // if TRUE, the instance afterwards gets moved into the copy code (online change)
END_VAR
AddInput('stValue', stValue);
AddInput('ipContainer', ipContainer);
AddInput('hrPrev', hrPrev);
AddOutput('ipContainer', ipContainer);
AddOutput('hresult',hresult);
END_METHOD

METHOD PUBLIC  Clone : I_Node
VAR
    pNode : POINTER TO Node_F_VN_AddToContainerElements_TcVnRotatedRectangle;
END_VAR
pNode := __NEW(Node_F_VN_AddToContainerElements_TcVnRotatedRectangle);
Clone := pNode^;
END_METHOD

METHOD PROTECTED OnExecute
hresult.Value := F_VN_AddToContainerElements_TcVnRotatedRectangle(
    stValue := stValue.Value,
    ipContainer := ipContainer.Value,
    hrPrev:= hrPrev.Value);
END_METHOD

METHOD PUBLIC PreExecutionCheck
VAR_INPUT
    Check : I_PreExecutionChecks;
END_VAR
Check.IsTrue(ipContainer.IsValid, 'ipContainer must be a valid container');
Check.IsTrue(ipContainer.IsType(TC_GLOBAL_CONST_LIST.ContainerType_Vector_TcVnRotatedRectangle), 'ipContainer contains incorrect type');
END_METHOD

END_FUNCTION_BLOCK

// Nodes/Algebraic Container Ops/AddTo/Node_F_VN_AddToContainerElements_TcVnVector2_DINT
{attribute 'linkalways'} 
{attribute 'no_explicit_call' := 'This FB is a CLASS and must be accessed using methods or properties'}
{attribute 'enable_dynamic_creation'}
FUNCTION_BLOCK Node_F_VN_AddToContainerElements_TcVnVector2_DINT EXTENDS VisionNode
VAR
    aValue : _TcVnVector2_DINT;
    ipContainer : _ITcVnContainer;
    hrPrev : _HRESULT(S_OK);
    hresult : _HRESULT(S_OK);
END_VAR

METHOD FB_init : BOOL
VAR_INPUT
    bInitRetains : BOOL; // if TRUE, the retain variables are initialized (warm start / cold start)
    bInCopyCode : BOOL;  // if TRUE, the instance afterwards gets moved into the copy code (online change)
END_VAR
AddInput('aValue', aValue);
AddInput('ipContainer', ipContainer);
AddInput('hrPrev', hrPrev);
AddOutput('ipContainer', ipContainer);
AddOutput('hresult',hresult);
END_METHOD

METHOD PUBLIC  Clone : I_Node
VAR
    pNode : POINTER TO Node_F_VN_AddToContainerElements_TcVnVector2_DINT;
END_VAR
pNode := __NEW(Node_F_VN_AddToContainerElements_TcVnVector2_DINT);
Clone := pNode^;
END_METHOD

METHOD PROTECTED OnExecute
hresult.Value := F_VN_AddToContainerElements_TcVnVector2_DINT(
    aValue := aValue.Value,
    ipContainer := ipContainer.Value,
    hrPrev:= hrPrev.Value);
END_METHOD

METHOD PUBLIC PreExecutionCheck
VAR_INPUT
    Check : I_PreExecutionChecks;
END_VAR
Check.IsTrue(ipContainer.IsValid, 'ipContainer must be a valid container');
Check.IsTrue(ipContainer.IsType(TC_GLOBAL_CONST_LIST.ContainerType_Vector_TcVnVector2_DINT), 'ipContainer contains incorrect type');
END_METHOD

END_FUNCTION_BLOCK

// Nodes/Algebraic Container Ops/AddTo/Node_F_VN_AddToContainerElements_TcVnVector2_INT
{attribute 'linkalways'} 
{attribute 'no_explicit_call' := 'This FB is a CLASS and must be accessed using methods or properties'}
{attribute 'enable_dynamic_creation'}
FUNCTION_BLOCK Node_F_VN_AddToContainerElements_TcVnVector2_INT EXTENDS VisionNode
VAR
    aValue : _TcVnVector2_INT;
    ipContainer : _ITcVnContainer;
    hrPrev : _HRESULT(S_OK);
    hresult : _HRESULT(S_OK);
END_VAR

METHOD FB_init : BOOL
VAR_INPUT
    bInitRetains : BOOL; // if TRUE, the retain variables are initialized (warm start / cold start)
    bInCopyCode : BOOL;  // if TRUE, the instance afterwards gets moved into the copy code (online change)
END_VAR
AddInput('aValue', aValue);
AddInput('ipContainer', ipContainer);
AddInput('hrPrev', hrPrev);
AddOutput('ipContainer', ipContainer);
AddOutput('hresult',hresult);
END_METHOD

METHOD PUBLIC  Clone : I_Node
VAR
    pNode : POINTER TO Node_F_VN_AddToContainerElements_TcVnVector2_INT;
END_VAR
pNode := __NEW(Node_F_VN_AddToContainerElements_TcVnVector2_INT);
Clone := pNode^;
END_METHOD

METHOD PROTECTED OnExecute
hresult.Value := F_VN_AddToContainerElements_TcVnVector2_INT(
    aValue := aValue.Value,
    ipContainer := ipContainer.Value,
    hrPrev:= hrPrev.Value);
END_METHOD

METHOD PUBLIC PreExecutionCheck
VAR_INPUT
    Check : I_PreExecutionChecks;
END_VAR
Check.IsTrue(ipContainer.IsValid, 'ipContainer must be a valid container');
Check.IsTrue(ipContainer.IsType(TC_GLOBAL_CONST_LIST.ContainerType_Vector_TcVnVector2_INT), 'ipContainer contains incorrect type');
END_METHOD

END_FUNCTION_BLOCK

// Nodes/Algebraic Container Ops/AddTo/Node_F_VN_AddToContainerElements_TcVnVector2_REAL
{attribute 'linkalways'} 
{attribute 'no_explicit_call' := 'This FB is a CLASS and must be accessed using methods or properties'}
{attribute 'enable_dynamic_creation'}
FUNCTION_BLOCK Node_F_VN_AddToContainerElements_TcVnVector2_REAL EXTENDS VisionNode
VAR
    aValue : _TcVnVector2_REAL;
    ipContainer : _ITcVnContainer;
    hrPrev : _HRESULT(S_OK);
    hresult : _HRESULT(S_OK);
END_VAR

METHOD FB_init : BOOL
VAR_INPUT
    bInitRetains : BOOL; // if TRUE, the retain variables are initialized (warm start / cold start)
    bInCopyCode : BOOL;  // if TRUE, the instance afterwards gets moved into the copy code (online change)
END_VAR
AddInput('aValue', aValue);
AddInput('ipContainer', ipContainer);
AddInput('hrPrev', hrPrev);
AddOutput('ipContainer', ipContainer);
AddOutput('hresult',hresult);
END_METHOD

METHOD PUBLIC  Clone : I_Node
VAR
    pNode : POINTER TO Node_F_VN_AddToContainerElements_TcVnVector2_REAL;
END_VAR
pNode := __NEW(Node_F_VN_AddToContainerElements_TcVnVector2_REAL);
Clone := pNode^;
END_METHOD

METHOD PROTECTED OnExecute
hresult.Value := F_VN_AddToContainerElements_TcVnVector2_REAL(
    aValue := aValue.Value,
    ipContainer := ipContainer.Value,
    hrPrev:= hrPrev.Value);
END_METHOD

METHOD PUBLIC PreExecutionCheck
VAR_INPUT
    Check : I_PreExecutionChecks;
END_VAR
Check.IsTrue(ipContainer.IsValid, 'ipContainer must be a valid container');
Check.IsTrue(ipContainer.IsType(TC_GLOBAL_CONST_LIST.ContainerType_Vector_TcVnVector2_REAL), 'ipContainer contains incorrect type');
END_METHOD

END_FUNCTION_BLOCK

// Nodes/Algebraic Container Ops/AddTo/Node_F_VN_AddToContainerElements_TcVnVector2_SINT
{attribute 'linkalways'} 
{attribute 'no_explicit_call' := 'This FB is a CLASS and must be accessed using methods or properties'}
{attribute 'enable_dynamic_creation'}
FUNCTION_BLOCK Node_F_VN_AddToContainerElements_TcVnVector2_SINT EXTENDS VisionNode
VAR
    aValue : _TcVnVector2_SINT;
    ipContainer : _ITcVnContainer;
    hrPrev : _HRESULT(S_OK);
    hresult : _HRESULT(S_OK);
END_VAR

METHOD FB_init : BOOL
VAR_INPUT
    bInitRetains : BOOL; // if TRUE, the retain variables are initialized (warm start / cold start)
    bInCopyCode : BOOL;  // if TRUE, the instance afterwards gets moved into the copy code (online change)
END_VAR
AddInput('aValue', aValue);
AddInput('ipContainer', ipContainer);
AddInput('hrPrev', hrPrev);
AddOutput('ipContainer', ipContainer);
AddOutput('hresult',hresult);
END_METHOD

METHOD PUBLIC  Clone : I_Node
VAR
    pNode : POINTER TO Node_F_VN_AddToContainerElements_TcVnVector2_SINT;
END_VAR
pNode := __NEW(Node_F_VN_AddToContainerElements_TcVnVector2_SINT);
Clone := pNode^;
END_METHOD

METHOD PROTECTED OnExecute
hresult.Value := F_VN_AddToContainerElements_TcVnVector2_SINT(
    aValue := aValue.Value,
    ipContainer := ipContainer.Value,
    hrPrev:= hrPrev.Value);
END_METHOD

METHOD PUBLIC PreExecutionCheck
VAR_INPUT
    Check : I_PreExecutionChecks;
END_VAR
Check.IsTrue(ipContainer.IsValid, 'ipContainer must be a valid container');
Check.IsTrue(ipContainer.IsType(TC_GLOBAL_CONST_LIST.ContainerType_Vector_TcVnVector2_SINT), 'ipContainer contains incorrect type');
END_METHOD

END_FUNCTION_BLOCK

// Nodes/Algebraic Container Ops/AddTo/Node_F_VN_AddToContainerElements_TcVnVector2_UINT
{attribute 'linkalways'} 
{attribute 'no_explicit_call' := 'This FB is a CLASS and must be accessed using methods or properties'}
{attribute 'enable_dynamic_creation'}
FUNCTION_BLOCK Node_F_VN_AddToContainerElements_TcVnVector2_UINT EXTENDS VisionNode
VAR
    aValue : _TcVnVector2_UINT;
    ipContainer : _ITcVnContainer;
    hrPrev : _HRESULT(S_OK);
    hresult : _HRESULT(S_OK);
END_VAR

METHOD FB_init : BOOL
VAR_INPUT
    bInitRetains : BOOL; // if TRUE, the retain variables are initialized (warm start / cold start)
    bInCopyCode : BOOL;  // if TRUE, the instance afterwards gets moved into the copy code (online change)
END_VAR
AddInput('aValue', aValue);
AddInput('ipContainer', ipContainer);
AddInput('hrPrev', hrPrev);
AddOutput('ipContainer', ipContainer);
AddOutput('hresult',hresult);
END_METHOD

METHOD PUBLIC  Clone : I_Node
VAR
    pNode : POINTER TO Node_F_VN_AddToContainerElements_TcVnVector2_UINT;
END_VAR
pNode := __NEW(Node_F_VN_AddToContainerElements_TcVnVector2_UINT);
Clone := pNode^;
END_METHOD

METHOD PROTECTED OnExecute
hresult.Value := F_VN_AddToContainerElements_TcVnVector2_UINT(
    aValue := aValue.Value,
    ipContainer := ipContainer.Value,
    hrPrev:= hrPrev.Value);
END_METHOD

METHOD PUBLIC PreExecutionCheck
VAR_INPUT
    Check : I_PreExecutionChecks;
END_VAR
Check.IsTrue(ipContainer.IsValid, 'ipContainer must be a valid container');
Check.IsTrue(ipContainer.IsType(TC_GLOBAL_CONST_LIST.ContainerType_Vector_TcVnVector2_UINT), 'ipContainer contains incorrect type');
END_METHOD

END_FUNCTION_BLOCK

// Nodes/Algebraic Container Ops/AddTo/Node_F_VN_AddToContainerElements_TcVnVector2_USINT
{attribute 'linkalways'} 
{attribute 'no_explicit_call' := 'This FB is a CLASS and must be accessed using methods or properties'}
{attribute 'enable_dynamic_creation'}
FUNCTION_BLOCK Node_F_VN_AddToContainerElements_TcVnVector2_USINT EXTENDS VisionNode
VAR
    aValue : _TcVnVector2_USINT;
    ipContainer : _ITcVnContainer;
    hrPrev : _HRESULT(S_OK);
    hresult : _HRESULT(S_OK);
END_VAR

METHOD FB_init : BOOL
VAR_INPUT
    bInitRetains : BOOL; // if TRUE, the retain variables are initialized (warm start / cold start)
    bInCopyCode : BOOL;  // if TRUE, the instance afterwards gets moved into the copy code (online change)
END_VAR
AddInput('aValue', aValue);
AddInput('ipContainer', ipContainer);
AddInput('hrPrev', hrPrev);
AddOutput('ipContainer', ipContainer);
AddOutput('hresult',hresult);
END_METHOD

METHOD PUBLIC  Clone : I_Node
VAR
    pNode : POINTER TO Node_F_VN_AddToContainerElements_TcVnVector2_USINT;
END_VAR
pNode := __NEW(Node_F_VN_AddToContainerElements_TcVnVector2_USINT);
Clone := pNode^;
END_METHOD

METHOD PROTECTED OnExecute
hresult.Value := F_VN_AddToContainerElements_TcVnVector2_USINT(
    aValue := aValue.Value,
    ipContainer := ipContainer.Value,
    hrPrev:= hrPrev.Value);
END_METHOD

METHOD PUBLIC PreExecutionCheck
VAR_INPUT
    Check : I_PreExecutionChecks;
END_VAR
Check.IsTrue(ipContainer.IsValid, 'ipContainer must be a valid container');
Check.IsTrue(ipContainer.IsType(TC_GLOBAL_CONST_LIST.ContainerType_Vector_TcVnVector2_USINT), 'ipContainer contains incorrect type');
END_METHOD

END_FUNCTION_BLOCK

// Nodes/Algebraic Container Ops/AddTo/Node_F_VN_AddToContainerElements_TcVnVector3_INT
{attribute 'linkalways'} 
{attribute 'no_explicit_call' := 'This FB is a CLASS and must be accessed using methods or properties'}
{attribute 'enable_dynamic_creation'}
FUNCTION_BLOCK Node_F_VN_AddToContainerElements_TcVnVector3_INT EXTENDS VisionNode
VAR
    aValue : _TcVnVector3_INT;
    ipContainer : _ITcVnContainer;
    hrPrev : _HRESULT(S_OK);
    hresult : _HRESULT(S_OK);
END_VAR

METHOD FB_init : BOOL
VAR_INPUT
    bInitRetains : BOOL; // if TRUE, the retain variables are initialized (warm start / cold start)
    bInCopyCode : BOOL;  // if TRUE, the instance afterwards gets moved into the copy code (online change)
END_VAR
AddInput('aValue', aValue);
AddInput('ipContainer', ipContainer);
AddInput('hrPrev', hrPrev);
AddOutput('ipContainer', ipContainer);
AddOutput('hresult',hresult);
END_METHOD

METHOD PUBLIC  Clone : I_Node
VAR
    pNode : POINTER TO Node_F_VN_AddToContainerElements_TcVnVector3_INT;
END_VAR
pNode := __NEW(Node_F_VN_AddToContainerElements_TcVnVector3_INT);
Clone := pNode^;
END_METHOD

METHOD PROTECTED OnExecute
hresult.Value := F_VN_AddToContainerElements_TcVnVector3_INT(
    aValue := aValue.Value,
    ipContainer := ipContainer.Value,
    hrPrev:= hrPrev.Value);
END_METHOD

METHOD PUBLIC PreExecutionCheck
VAR_INPUT
    Check : I_PreExecutionChecks;
END_VAR
Check.IsTrue(ipContainer.IsValid, 'ipContainer must be a valid container');
Check.IsTrue(ipContainer.IsType(TC_GLOBAL_CONST_LIST.ContainerType_Vector_TcVnVector3_INT), 'ipContainer contains incorrect type');
END_METHOD

END_FUNCTION_BLOCK

// Nodes/Algebraic Container Ops/AddTo/Node_F_VN_AddToContainerElements_TcVnVector3_REAL
{attribute 'linkalways'} 
{attribute 'no_explicit_call' := 'This FB is a CLASS and must be accessed using methods or properties'}
{attribute 'enable_dynamic_creation'}
FUNCTION_BLOCK Node_F_VN_AddToContainerElements_TcVnVector3_REAL EXTENDS VisionNode
VAR
    aValue : _TcVnVector3_REAL;
    ipContainer : _ITcVnContainer;
    hrPrev : _HRESULT(S_OK);
    hresult : _HRESULT(S_OK);
END_VAR

METHOD FB_init : BOOL
VAR_INPUT
    bInitRetains : BOOL; // if TRUE, the retain variables are initialized (warm start / cold start)
    bInCopyCode : BOOL;  // if TRUE, the instance afterwards gets moved into the copy code (online change)
END_VAR
AddInput('aValue', aValue);
AddInput('ipContainer', ipContainer);
AddInput('hrPrev', hrPrev);
AddOutput('ipContainer', ipContainer);
AddOutput('hresult',hresult);
END_METHOD

METHOD PUBLIC  Clone : I_Node
VAR
    pNode : POINTER TO Node_F_VN_AddToContainerElements_TcVnVector3_REAL;
END_VAR
pNode := __NEW(Node_F_VN_AddToContainerElements_TcVnVector3_REAL);
Clone := pNode^;
END_METHOD

METHOD PROTECTED OnExecute
hresult.Value := F_VN_AddToContainerElements_TcVnVector3_REAL(
    aValue := aValue.Value,
    ipContainer := ipContainer.Value,
    hrPrev:= hrPrev.Value);
END_METHOD

METHOD PUBLIC PreExecutionCheck
VAR_INPUT
    Check : I_PreExecutionChecks;
END_VAR
Check.IsTrue(ipContainer.IsValid, 'ipContainer must be a valid container');
Check.IsTrue(ipContainer.IsType(TC_GLOBAL_CONST_LIST.ContainerType_Vector_TcVnVector3_REAL), 'ipContainer contains incorrect type');
END_METHOD

END_FUNCTION_BLOCK

// Nodes/Algebraic Container Ops/AddTo/Node_F_VN_AddToContainerElements_TcVnVector3_SINT
{attribute 'linkalways'} 
{attribute 'no_explicit_call' := 'This FB is a CLASS and must be accessed using methods or properties'}
{attribute 'enable_dynamic_creation'}
FUNCTION_BLOCK Node_F_VN_AddToContainerElements_TcVnVector3_SINT EXTENDS VisionNode
VAR
    aValue : _TcVnVector3_SINT;
    ipContainer : _ITcVnContainer;
    hrPrev : _HRESULT(S_OK);
    hresult : _HRESULT(S_OK);
END_VAR

METHOD FB_init : BOOL
VAR_INPUT
    bInitRetains : BOOL; // if TRUE, the retain variables are initialized (warm start / cold start)
    bInCopyCode : BOOL;  // if TRUE, the instance afterwards gets moved into the copy code (online change)
END_VAR
AddInput('aValue', aValue);
AddInput('ipContainer', ipContainer);
AddInput('hrPrev', hrPrev);
AddOutput('ipContainer', ipContainer);
AddOutput('hresult',hresult);
END_METHOD

METHOD PUBLIC  Clone : I_Node
VAR
    pNode : POINTER TO Node_F_VN_AddToContainerElements_TcVnVector3_SINT;
END_VAR
pNode := __NEW(Node_F_VN_AddToContainerElements_TcVnVector3_SINT);
Clone := pNode^;
END_METHOD

METHOD PROTECTED OnExecute
hresult.Value := F_VN_AddToContainerElements_TcVnVector3_SINT(
    aValue := aValue.Value,
    ipContainer := ipContainer.Value,
    hrPrev:= hrPrev.Value);
END_METHOD

METHOD PUBLIC PreExecutionCheck
VAR_INPUT
    Check : I_PreExecutionChecks;
END_VAR
Check.IsTrue(ipContainer.IsValid, 'ipContainer must be a valid container');
Check.IsTrue(ipContainer.IsType(TC_GLOBAL_CONST_LIST.ContainerType_Vector_TcVnVector3_SINT), 'ipContainer contains incorrect type');
END_METHOD

END_FUNCTION_BLOCK

// Nodes/Algebraic Container Ops/AddTo/Node_F_VN_AddToContainerElements_TcVnVector3_UINT
{attribute 'linkalways'} 
{attribute 'no_explicit_call' := 'This FB is a CLASS and must be accessed using methods or properties'}
{attribute 'enable_dynamic_creation'}
FUNCTION_BLOCK Node_F_VN_AddToContainerElements_TcVnVector3_UINT EXTENDS VisionNode
VAR
    aValue : _TcVnVector3_UINT;
    ipContainer : _ITcVnContainer;
    hrPrev : _HRESULT(S_OK);
    hresult : _HRESULT(S_OK);
END_VAR

METHOD FB_init : BOOL
VAR_INPUT
    bInitRetains : BOOL; // if TRUE, the retain variables are initialized (warm start / cold start)
    bInCopyCode : BOOL;  // if TRUE, the instance afterwards gets moved into the copy code (online change)
END_VAR
AddInput('aValue', aValue);
AddInput('ipContainer', ipContainer);
AddInput('hrPrev', hrPrev);
AddOutput('ipContainer', ipContainer);
AddOutput('hresult',hresult);
END_METHOD

METHOD PUBLIC  Clone : I_Node
VAR
    pNode : POINTER TO Node_F_VN_AddToContainerElements_TcVnVector3_UINT;
END_VAR
pNode := __NEW(Node_F_VN_AddToContainerElements_TcVnVector3_UINT);
Clone := pNode^;
END_METHOD

METHOD PROTECTED OnExecute
hresult.Value := F_VN_AddToContainerElements_TcVnVector3_UINT(
    aValue := aValue.Value,
    ipContainer := ipContainer.Value,
    hrPrev:= hrPrev.Value);
END_METHOD

METHOD PUBLIC PreExecutionCheck
VAR_INPUT
    Check : I_PreExecutionChecks;
END_VAR
Check.IsTrue(ipContainer.IsValid, 'ipContainer must be a valid container');
Check.IsTrue(ipContainer.IsType(TC_GLOBAL_CONST_LIST.ContainerType_Vector_TcVnVector3_UINT), 'ipContainer contains incorrect type');
END_METHOD

END_FUNCTION_BLOCK

// Nodes/Algebraic Container Ops/AddTo/Node_F_VN_AddToContainerElements_TcVnVector3_USINT
{attribute 'linkalways'} 
{attribute 'no_explicit_call' := 'This FB is a CLASS and must be accessed using methods or properties'}
{attribute 'enable_dynamic_creation'}
FUNCTION_BLOCK Node_F_VN_AddToContainerElements_TcVnVector3_USINT EXTENDS VisionNode
VAR
    aValue : _TcVnVector3_USINT;
    ipContainer : _ITcVnContainer;
    hrPrev : _HRESULT(S_OK);
    hresult : _HRESULT(S_OK);
END_VAR

METHOD FB_init : BOOL
VAR_INPUT
    bInitRetains : BOOL; // if TRUE, the retain variables are initialized (warm start / cold start)
    bInCopyCode : BOOL;  // if TRUE, the instance afterwards gets moved into the copy code (online change)
END_VAR
AddInput('aValue', aValue);
AddInput('ipContainer', ipContainer);
AddInput('hrPrev', hrPrev);
AddOutput('ipContainer', ipContainer);
AddOutput('hresult',hresult);
END_METHOD

METHOD PUBLIC  Clone : I_Node
VAR
    pNode : POINTER TO Node_F_VN_AddToContainerElements_TcVnVector3_USINT;
END_VAR
pNode := __NEW(Node_F_VN_AddToContainerElements_TcVnVector3_USINT);
Clone := pNode^;
END_METHOD

METHOD PROTECTED OnExecute
hresult.Value := F_VN_AddToContainerElements_TcVnVector3_USINT(
    aValue := aValue.Value,
    ipContainer := ipContainer.Value,
    hrPrev:= hrPrev.Value);
END_METHOD

METHOD PUBLIC PreExecutionCheck
VAR_INPUT
    Check : I_PreExecutionChecks;
END_VAR
Check.IsTrue(ipContainer.IsValid, 'ipContainer must be a valid container');
Check.IsTrue(ipContainer.IsType(TC_GLOBAL_CONST_LIST.ContainerType_Vector_TcVnVector3_USINT), 'ipContainer contains incorrect type');
END_METHOD

END_FUNCTION_BLOCK

// Nodes/Algebraic Container Ops/AddTo/Node_F_VN_AddToContainerElements_TcVnVector4_DINT
{attribute 'linkalways'} 
{attribute 'no_explicit_call' := 'This FB is a CLASS and must be accessed using methods or properties'}
{attribute 'enable_dynamic_creation'}
FUNCTION_BLOCK Node_F_VN_AddToContainerElements_TcVnVector4_DINT EXTENDS VisionNode
VAR
    aValue : _TcVnVector4_DINT;
    ipContainer : _ITcVnContainer;
    hrPrev : _HRESULT(S_OK);
    hresult : _HRESULT(S_OK);
END_VAR

METHOD FB_init : BOOL
VAR_INPUT
    bInitRetains : BOOL; // if TRUE, the retain variables are initialized (warm start / cold start)
    bInCopyCode : BOOL;  // if TRUE, the instance afterwards gets moved into the copy code (online change)
END_VAR
AddInput('aValue', aValue);
AddInput('ipContainer', ipContainer);
AddInput('hrPrev', hrPrev);
AddOutput('ipContainer', ipContainer);
AddOutput('hresult',hresult);
END_METHOD

METHOD PUBLIC  Clone : I_Node
VAR
    pNode : POINTER TO Node_F_VN_AddToContainerElements_TcVnVector4_DINT;
END_VAR
pNode := __NEW(Node_F_VN_AddToContainerElements_TcVnVector4_DINT);
Clone := pNode^;
END_METHOD

METHOD PROTECTED OnExecute
hresult.Value := F_VN_AddToContainerElements_TcVnVector4_DINT(
    aValue := aValue.Value,
    ipContainer := ipContainer.Value,
    hrPrev:= hrPrev.Value);
END_METHOD

METHOD PUBLIC PreExecutionCheck
VAR_INPUT
    Check : I_PreExecutionChecks;
END_VAR
Check.IsTrue(ipContainer.IsValid, 'ipContainer must be a valid container');
Check.IsTrue(ipContainer.IsType(TC_GLOBAL_CONST_LIST.ContainerType_Vector_TcVnVector4_DINT), 'ipContainer contains incorrect type');
END_METHOD

END_FUNCTION_BLOCK

// Nodes/Algebraic Container Ops/AddTo/Node_F_VN_AddToContainerElements_TcVnVector4_INT
{attribute 'linkalways'} 
{attribute 'no_explicit_call' := 'This FB is a CLASS and must be accessed using methods or properties'}
{attribute 'enable_dynamic_creation'}
FUNCTION_BLOCK Node_F_VN_AddToContainerElements_TcVnVector4_INT EXTENDS VisionNode
VAR
    aValue : _TcVnVector4_INT;
    ipContainer : _ITcVnContainer;
    hrPrev : _HRESULT(S_OK);
    hresult : _HRESULT(S_OK);
END_VAR

METHOD FB_init : BOOL
VAR_INPUT
    bInitRetains : BOOL; // if TRUE, the retain variables are initialized (warm start / cold start)
    bInCopyCode : BOOL;  // if TRUE, the instance afterwards gets moved into the copy code (online change)
END_VAR
AddInput('aValue', aValue);
AddInput('ipContainer', ipContainer);
AddInput('hrPrev', hrPrev);
AddOutput('ipContainer', ipContainer);
AddOutput('hresult',hresult);
END_METHOD

METHOD PUBLIC  Clone : I_Node
VAR
    pNode : POINTER TO Node_F_VN_AddToContainerElements_TcVnVector4_INT;
END_VAR
pNode := __NEW(Node_F_VN_AddToContainerElements_TcVnVector4_INT);
Clone := pNode^;
END_METHOD

METHOD PROTECTED OnExecute
hresult.Value := F_VN_AddToContainerElements_TcVnVector4_INT(
    aValue := aValue.Value,
    ipContainer := ipContainer.Value,
    hrPrev:= hrPrev.Value);
END_METHOD

METHOD PUBLIC PreExecutionCheck
VAR_INPUT
    Check : I_PreExecutionChecks;
END_VAR
Check.IsTrue(ipContainer.IsValid, 'ipContainer must be a valid container');
Check.IsTrue(ipContainer.IsType(TC_GLOBAL_CONST_LIST.ContainerType_Vector_TcVnVector4_INT), 'ipContainer contains incorrect type');
END_METHOD

END_FUNCTION_BLOCK

// Nodes/Algebraic Container Ops/AddTo/Node_F_VN_AddToContainerElements_TcVnVector4_LREAL
{attribute 'linkalways'} 
{attribute 'no_explicit_call' := 'This FB is a CLASS and must be accessed using methods or properties'}
{attribute 'enable_dynamic_creation'}
FUNCTION_BLOCK Node_F_VN_AddToContainerElements_TcVnVector4_LREAL EXTENDS VisionNode
VAR
    aValue : _TcVnVector4_LREAL;
    ipContainer : _ITcVnContainer;
    hrPrev : _HRESULT(S_OK);
    hresult : _HRESULT(S_OK);
END_VAR

METHOD FB_init : BOOL
VAR_INPUT
    bInitRetains : BOOL; // if TRUE, the retain variables are initialized (warm start / cold start)
    bInCopyCode : BOOL;  // if TRUE, the instance afterwards gets moved into the copy code (online change)
END_VAR
AddInput('aValue', aValue);
AddInput('ipContainer', ipContainer);
AddInput('hrPrev', hrPrev);
AddOutput('ipContainer', ipContainer);
AddOutput('hresult',hresult);
END_METHOD

METHOD PUBLIC  Clone : I_Node
VAR
    pNode : POINTER TO Node_F_VN_AddToContainerElements_TcVnVector4_LREAL;
END_VAR
pNode := __NEW(Node_F_VN_AddToContainerElements_TcVnVector4_LREAL);
Clone := pNode^;
END_METHOD

METHOD PROTECTED OnExecute
hresult.Value := F_VN_AddToContainerElements_TcVnVector4_LREAL(
    aValue := aValue.Value,
    ipContainer := ipContainer.Value,
    hrPrev:= hrPrev.Value);
END_METHOD

METHOD PUBLIC PreExecutionCheck
VAR_INPUT
    Check : I_PreExecutionChecks;
END_VAR
Check.IsTrue(ipContainer.IsValid, 'ipContainer must be a valid container');
Check.IsTrue(ipContainer.IsType(TC_GLOBAL_CONST_LIST.ContainerType_Vector_TcVnVector4_LREAL), 'ipContainer contains incorrect type');
END_METHOD

END_FUNCTION_BLOCK

// Nodes/Algebraic Container Ops/AddTo/Node_F_VN_AddToContainerElements_TcVnVector4_REAL
{attribute 'linkalways'} 
{attribute 'no_explicit_call' := 'This FB is a CLASS and must be accessed using methods or properties'}
{attribute 'enable_dynamic_creation'}
FUNCTION_BLOCK Node_F_VN_AddToContainerElements_TcVnVector4_REAL EXTENDS VisionNode
VAR
    aValue : _TcVnVector4_REAL;
    ipContainer : _ITcVnContainer;
    hrPrev : _HRESULT(S_OK);
    hresult : _HRESULT(S_OK);
END_VAR

METHOD FB_init : BOOL
VAR_INPUT
    bInitRetains : BOOL; // if TRUE, the retain variables are initialized (warm start / cold start)
    bInCopyCode : BOOL;  // if TRUE, the instance afterwards gets moved into the copy code (online change)
END_VAR
AddInput('aValue', aValue);
AddInput('ipContainer', ipContainer);
AddInput('hrPrev', hrPrev);
AddOutput('ipContainer', ipContainer);
AddOutput('hresult',hresult);
END_METHOD

METHOD PUBLIC  Clone : I_Node
VAR
    pNode : POINTER TO Node_F_VN_AddToContainerElements_TcVnVector4_REAL;
END_VAR
pNode := __NEW(Node_F_VN_AddToContainerElements_TcVnVector4_REAL);
Clone := pNode^;
END_METHOD

METHOD PROTECTED OnExecute
hresult.Value := F_VN_AddToContainerElements_TcVnVector4_REAL(
    aValue := aValue.Value,
    ipContainer := ipContainer.Value,
    hrPrev:= hrPrev.Value);
END_METHOD

METHOD PUBLIC PreExecutionCheck
VAR_INPUT
    Check : I_PreExecutionChecks;
END_VAR
Check.IsTrue(ipContainer.IsValid, 'ipContainer must be a valid container');
Check.IsTrue(ipContainer.IsType(TC_GLOBAL_CONST_LIST.ContainerType_Vector_TcVnVector4_REAL), 'ipContainer contains incorrect type');
END_METHOD

END_FUNCTION_BLOCK

// Nodes/Algebraic Container Ops/AddTo/Node_F_VN_AddToContainerElements_TcVnVector4_SINT
{attribute 'linkalways'} 
{attribute 'no_explicit_call' := 'This FB is a CLASS and must be accessed using methods or properties'}
{attribute 'enable_dynamic_creation'}
FUNCTION_BLOCK Node_F_VN_AddToContainerElements_TcVnVector4_SINT EXTENDS VisionNode
VAR
    aValue : _TcVnVector4_SINT;
    ipContainer : _ITcVnContainer;
    hrPrev : _HRESULT(S_OK);
    hresult : _HRESULT(S_OK);
END_VAR

METHOD FB_init : BOOL
VAR_INPUT
    bInitRetains : BOOL; // if TRUE, the retain variables are initialized (warm start / cold start)
    bInCopyCode : BOOL;  // if TRUE, the instance afterwards gets moved into the copy code (online change)
END_VAR
AddInput('aValue', aValue);
AddInput('ipContainer', ipContainer);
AddInput('hrPrev', hrPrev);
AddOutput('ipContainer', ipContainer);
AddOutput('hresult',hresult);
END_METHOD

METHOD PUBLIC  Clone : I_Node
VAR
    pNode : POINTER TO Node_F_VN_AddToContainerElements_TcVnVector4_SINT;
END_VAR
pNode := __NEW(Node_F_VN_AddToContainerElements_TcVnVector4_SINT);
Clone := pNode^;
END_METHOD

METHOD PROTECTED OnExecute
hresult.Value := F_VN_AddToContainerElements_TcVnVector4_SINT(
    aValue := aValue.Value,
    ipContainer := ipContainer.Value,
    hrPrev:= hrPrev.Value);
END_METHOD

METHOD PUBLIC PreExecutionCheck
VAR_INPUT
    Check : I_PreExecutionChecks;
END_VAR
Check.IsTrue(ipContainer.IsValid, 'ipContainer must be a valid container');
Check.IsTrue(ipContainer.IsType(TC_GLOBAL_CONST_LIST.ContainerType_Vector_TcVnVector4_SINT), 'ipContainer contains incorrect type');
END_METHOD

END_FUNCTION_BLOCK

